LIN {X 0,Y 421.883,Z 601.374,A -85,B 0,C 180,E1 -10153.456,E2 -10153.456} C_VEL
LIN {X 0,Y 421.234,Z 614.501,A -85,B 0,C 180,E1 -10153.897,E2 -10153.897} C_VEL
LIN {X 0,Y 420.74,Z 626.729,A -85,B 0,C 180,E1 -10154.499,E2 -10154.499} C_VEL
LIN {X 0,Y 419.97,Z 639.362,A -85,B 0,C 180,E1 -10155.339,E2 -10155.339} C_VEL
LIN {X 0,Y 419.355,Z 650.7,A -85,B 0,C 180,E1 -10156.307,E2 -10156.307} C_VEL
LIN {X 0,Y 418.794,Z 660.932,A -85,B 0,C 180,E1 -10157.399,E2 -10157.399} C_VEL
LIN {X 0,Y 418.224,Z 670.168,A -85,B 0,C 180,E1 -10158.612,E2 -10158.612} C_VEL
LIN {X 0,Y 417.717,Z 679.182,A -85,B 0,C 180,E1 -10160.07,E2 -10160.07} C_VEL
LIN {X 0,Y 417.45,Z 686.381,A -85,B 0,C 180,E1 -10161.529,E2 -10161.529} C_VEL
LIN {X 0,Y 417.234,Z 692.934,A -85,B 0,C 180,E1 -10163.229,E2 -10163.229} C_VEL
LIN {X 0,Y 417.235,Z 697.222,A -85,B 0,C 180,E1 -10164.685,E2 -10164.685} C_VEL
LIN {X 0,Y 417.147,Z 700.376,A -85,B 0,C 180,E1 -10166.136,E2 -10166.136} C_VEL
LIN {X 0,Y 417.232,Z 701.935,A -85,B 0,C 180,E1 -10167.104,E2 -10167.104} C_VEL
LIN {X 0,Y 417.247,Z 703.007,A -85,B 0,C 180,E1 -10168.07,E2 -10168.07} C_VEL
LIN {X 0,Y 417.206,Z 703.65,A -85,B 0,C 180,E1 -10169.035,E2 -10169.035} C_VEL
LIN {X 0,Y 417.179,Z 703.882,A -85,B 0,C 180,E1 -10170,E2 -10170} C_VEL
LIN {X 0,Y 417.207,Z 703.694,A -85,B 0,C 180,E1 -10170.966,E2 -10170.966} C_VEL
LIN {X 0,Y 417.238,Z 703.046,A -85,B 0,C 180,E1 -10171.931,E2 -10171.931} C_VEL
LIN {X 0,Y 417.242,Z 701.982,A -85,B 0,C 180,E1 -10172.897,E2 -10172.897} C_VEL
LIN {X 0,Y 417.146,Z 700.49,A -85,B 0,C 180,E1 -10173.865,E2 -10173.865} C_VEL
LIN {X 0,Y 417.197,Z 697.385,A -85,B 0,C 180,E1 -10175.317,E2 -10175.317} C_VEL
LIN {X 0,Y 417.243,Z 693.186,A -85,B 0,C 180,E1 -10176.772,E2 -10176.772} C_VEL
LIN {X 0,Y 417.448,Z 686.754,A -85,B 0,C 180,E1 -10178.472,E2 -10178.472} C_VEL
LIN {X 0,Y 417.762,Z 679.755,A -85,B 0,C 180,E1 -10179.93,E2 -10179.93} C_VEL
LIN {X 0,Y 418.247,Z 671.097,A -85,B 0,C 180,E1 -10181.388,E2 -10181.388} C_VEL
LIN {X 0,Y 418.776,Z 662.214,A -85,B 0,C 180,E1 -10182.602,E2 -10182.602} C_VEL
LIN {X 0,Y 419.488,Z 651.309,A -85,B 0,C 180,E1 -10183.813,E2 -10183.813} C_VEL
LIN {X 0,Y 420.239,Z 640.549,A -85,B 0,C 180,E1 -10184.776,E2 -10184.776} C_VEL
LIN {X 0,Y 421.009,Z 628.693,A -85,B 0,C 180,E1 -10185.616,E2 -10185.616} C_VEL
LIN {X 0,Y 421.731,Z 615.268,A -85,B 0,C 180,E1 -10186.333,E2 -10186.333} C_VEL
LIN {X 0,Y 422.424,Z 602.737,A -85,B 0,C 180,E1 -10186.803,E2 -10186.803} C_VEL
LIN {X 0,Y 422.79,Z 586.028,A -85,B 0,C 180,E1 -10187.192,E2 -10187.192} C_VEL
LIN {X 0,Y 423.985,Z 519.859,A -85,B 0,C 180,E1 -10188.527,E2 -10188.527} C_VEL
LIN {X 0,Y 421.419,Z 498.098,A -85,B 0,C 180,E1 -10189.145,E2 -10189.145} C_VEL
LIN {X 0,Y 419.729,Z 487.424,A -85,B 0,C 180,E1 -10189.496,E2 -10189.496} C_VEL
LIN {X 0,Y 420.98,Z 467.923,A -85,B 0,C 180,E1 -10192.98,E2 -10192.98} C_VEL
LIN {X 0,Y 422.264,Z 451.431,A -85,B 0,C 180,E1 -10196.005,E2 -10196.005} C_VEL
LIN {X 0,Y 421.657,Z 446.488,A -85,B 0,C 180,E1 -10197.001,E2 -10197.001} C_VEL
LIN {X 0,Y 419.324,Z 435.566,A -85,B 0,C 180,E1 -10199.362,E2 -10199.362} C_VEL
LIN {X 0,Y 418.269,Z 431.387,A -85,B 0,C 180,E1 -10200.331,E2 -10200.331} C_VEL
LIN {X 0,Y 418.252,Z 431.392,A -85,B 0,C 180,E1 -10203.677,E2 -10203.677} C_VEL
LIN {X 0,Y 418.244,Z 431.39,A -85,B 0,C 180,E1 -10207.224,E2 -10207.224} C_VEL
LIN {X 0,Y 418.255,Z 431.385,A -85,B 0,C 180,E1 -10209.682,E2 -10209.682} C_VEL
LIN {X 0,Y 418.233,Z 431.388,A -85,B 0,C 180,E1 -10212.321,E2 -10212.321} C_VEL
LIN {X 0,Y 418.239,Z 431.387,A -85,B 0,C 180,E1 -10215.109,E2 -10215.109} C_VEL
LIN {X 0,Y 418.238,Z 431.385,A -85,B 0,C 180,E1 -10217.766,E2 -10217.766} C_VEL
LIN {X 0,Y 418.246,Z 431.388,A -85,B 0,C 180,E1 -10220.621,E2 -10220.621} C_VEL
LIN {X 0,Y 418.246,Z 431.384,A -85,B 0,C 180,E1 -10223.976,E2 -10223.976} C_VEL
LIN {X 0,Y 418.261,Z 431.381,A -85,B 0,C 180,E1 -10227.156,E2 -10227.156} C_VEL
LIN {X 0,Y 418.262,Z 431.384,A -85,B 0,C 180,E1 -10230.838,E2 -10230.838} C_VEL
LIN {X 0,Y 418.229,Z 431.388,A -85,B 0,C 180,E1 -10234.093,E2 -10234.093} C_VEL
LIN {X 0,Y 418.231,Z 431.387,A -85,B 0,C 180,E1 -10237.263,E2 -10237.263} C_VEL
LIN {X 0,Y 418.248,Z 431.388,A -85,B 0,C 180,E1 -10240.362,E2 -10240.362} C_VEL
LIN {X 0,Y 418.283,Z 431.381,A -85,B 0,C 180,E1 -10243.403,E2 -10243.403} C_VEL
LIN {X 0,Y 418.348,Z 431.374,A -85,B 0,C 180,E1 -10247.385,E2 -10247.385} C_VEL
LIN {X 0,Y 418.369,Z 431.373,A -85,B 0,C 180,E1 -10251.304,E2 -10251.304} C_VEL
LIN {X 0,Y 418.445,Z 431.365,A -85,B 0,C 180,E1 -10254.518,E2 -10254.518} C_VEL
LIN {X 0,Y 418.966,Z 434.693,A -85,B 0,C 180,E1 -10255.568,E2 -10255.568} C_VEL
LIN {X 0,Y 424.854,Z 448.746,A -85,B 0,C 180,E1 -10256.248,E2 -10256.248} C_VEL
LIN {X 0,Y 423.209,Z 531.742,A -85,B 0,C 180,E1 -10257.952,E2 -10257.952} C_VEL
LIN {X 0,Y 422.943,Z 545.326,A -85,B 0,C 180,E1 -10258.304,E2 -10258.304} C_VEL
LIN {X 0,Y 422.569,Z 558.852,A -85,B 0,C 180,E1 -10258.868,E2 -10258.868} C_VEL
LIN {X 0,Y 422.136,Z 570.169,A -85,B 0,C 180,E1 -10259.519,E2 -10259.519} C_VEL
LIN {X 0,Y 421.493,Z 580.942,A -85,B 0,C 180,E1 -10260.312,E2 -10260.312} C_VEL
LIN {X 0,Y 420.713,Z 592.908,A -85,B 0,C 180,E1 -10261.436,E2 -10261.436} C_VEL
LIN {X 0,Y 420.173,Z 601.191,A -85,B 0,C 180,E1 -10262.397,E2 -10262.397} C_VEL
LIN {X 0,Y 419.534,Z 609.83,A -85,B 0,C 180,E1 -10263.602,E2 -10263.602} C_VEL
LIN {X 0,Y 418.92,Z 618.208,A -85,B 0,C 180,E1 -10265.053,E2 -10265.053} C_VEL
LIN {X 0,Y 418.49,Z 624.908,A -85,B 0,C 180,E1 -10266.509,E2 -10266.509} C_VEL
LIN {X 0,Y 418.087,Z 629.473,A -85,B 0,C 180,E1 -10267.728,E2 -10267.728} C_VEL
LIN {X 0,Y 417.78,Z 633.809,A -85,B 0,C 180,E1 -10269.196,E2 -10269.196} C_VEL
LIN {X 0,Y 417.51,Z 637.049,A -85,B 0,C 180,E1 -10270.671,E2 -10270.671} C_VEL
LIN {X 0,Y 417.341,Z 639.511,A -85,B 0,C 180,E1 -10272.386,E2 -10272.386} C_VEL
LIN {X 0,Y 417.209,Z 640.47,A -85,B 0,C 180,E1 -10273.641,E2 -10273.641} C_VEL
LIN {X 0,Y 417.175,Z 640.732,A -85,B 0,C 180,E1 -10274.637,E2 -10274.637} C_VEL
LIN {X 0,Y 417.198,Z 640.252,A -85,B 0,C 180,E1 -10276.216,E2 -10276.216} C_VEL
LIN {X 0,Y 417.235,Z 638.852,A -85,B 0,C 180,E1 -10277.65,E2 -10277.65} C_VEL
LIN {X 0,Y 417.336,Z 637.328,A -85,B 0,C 180,E1 -10278.661,E2 -10278.661} C_VEL
LIN {X 0,Y 417.508,Z 634.078,A -85,B 0,C 180,E1 -10280.187,E2 -10280.187} C_VEL
LIN {X 0,Y 417.735,Z 629.594,A -85,B 0,C 180,E1 -10281.724,E2 -10281.724} C_VEL
LIN {X 0,Y 418.055,Z 623.72,A -85,B 0,C 180,E1 -10283.27,E2 -10283.27} C_VEL
LIN {X 0,Y 418.516,Z 616.248,A -85,B 0,C 180,E1 -10284.823,E2 -10284.823} C_VEL
LIN {X 0,Y 418.986,Z 608.45,A -85,B 0,C 180,E1 -10286.124,E2 -10286.124} C_VEL
LIN {X 0,Y 419.606,Z 598.921,A -85,B 0,C 180,E1 -10287.414,E2 -10287.414} C_VEL
LIN {X 0,Y 420.198,Z 588.06,A -85,B 0,C 180,E1 -10288.605,E2 -10288.605} C_VEL
LIN {X 0,Y 420.853,Z 576.14,A -85,B 0,C 180,E1 -10289.63,E2 -10289.63} C_VEL
LIN {X 0,Y 421.373,Z 564.13,A -85,B 0,C 180,E1 -10290.439,E2 -10290.439} C_VEL
LIN {X 0,Y 421.814,Z 551.719,A -85,B 0,C 180,E1 -10291.063,E2 -10291.063} C_VEL
LIN {X 0,Y 422.135,Z 538.458,A -85,B 0,C 180,E1 -10291.523,E2 -10291.523} C_VEL
LIN {X 0,Y 422.624,Z 503.985,A -85,B 0,C 180,E1 -10292.209,E2 -10292.209} C_VEL
LIN {X 0,Y 423.54,Z 447.206,A -85,B 0,C 180,E1 -10293.307,E2 -10293.307} C_VEL
LIN {X 0,Y 418.282,Z 431.382,A -85,B 0,C 180,E1 -10293.868,E2 -10293.868} C_VEL
LIN {X 0,Y 418.237,Z 431.383,A -85,B 0,C 180,E1 -10297.225,E2 -10297.225} C_VEL
LIN {X 0,Y 418.21,Z 431.389,A -85,B 0,C 180,E1 -10300.867,E2 -10300.867} C_VEL
LIN {X 0,Y 418.206,Z 431.388,A -85,B 0,C 180,E1 -10303.728,E2 -10303.728} C_VEL
LIN {X 0,Y 418.202,Z 431.395,A -85,B 0,C 180,E1 -10306.447,E2 -10306.447} C_VEL
LIN {X 0,Y 418.209,Z 431.387,A -85,B 0,C 180,E1 -10309.133,E2 -10309.133} C_VEL
LIN {X 0,Y 418.235,Z 431.387,A -85,B 0,C 180,E1 -10312.775,E2 -10312.775} C_VEL
LIN {X 0,Y 418.25,Z 431.388,A -85,B 0,C 180,E1 -10316.323,E2 -10316.323} C_VEL
LIN {X 0,Y 418.243,Z 431.383,A -85,B 0,C 180,E1 -10319.727,E2 -10319.727} C_VEL
LIN {X 0,Y 418.219,Z 431.387,A -85,B 0,C 180,E1 -10323.017,E2 -10323.017} C_VEL
LIN {X 0,Y 418.286,Z 431.382,A -85,B 0,C 180,E1 -10326.218,E2 -10326.218} C_VEL
LIN {X 0,Y 418.252,Z 431.381,A -85,B 0,C 180,E1 -10329.337,E2 -10329.337} C_VEL
LIN {X 0,Y 418.279,Z 431.385,A -85,B 0,C 180,E1 -10332.395,E2 -10332.395} C_VEL
LIN {X 0,Y 418.3,Z 431.375,A -85,B 0,C 180,E1 -10335.403,E2 -10335.403} C_VEL
LIN {X 0,Y 418.316,Z 431.38,A -85,B 0,C 180,E1 -10338.369,E2 -10338.369} C_VEL
LIN {X 0,Y 418.379,Z 431.366,A -85,B 0,C 180,E1 -10341.304,E2 -10341.304} C_VEL
LIN {X 0,Y 418.491,Z 431.356,A -85,B 0,C 180,E1 -10344.217,E2 -10344.217} C_VEL
LIN {X 0,Y 418.366,Z 431.367,A -85,B 0,C 180,E1 -10344.893,E2 -10344.893} C_VEL
LIN {X 0,Y 417.623,Z 431.461,A -85,B 0,C 180,E1 -10345.697,E2 -10345.697} C_VEL
LIN {X 0,Y 414.751,Z 431.821,A -85,B 0,C 180,E1 -10347.005,E2 -10347.005} C_VEL
LIN {X 0,Y 412.417,Z 432.112,A -85,B 0,C 180,E1 -10348.061,E2 -10348.061} C_VEL
LIN {X 0,Y 411.491,Z 432.227,A -85,B 0,C 180,E1 -10348.877,E2 -10348.877} C_VEL
LIN {X 0,Y 411.452,Z 432.229,A -85,B 0,C 180,E1 -10349.152,E2 -10349.152} C_VEL
LIN {X 0,Y 411.635,Z 432.208,A -85,B 0,C 180,E1 -10350,E2 -10350} C_VEL
LIN {X 0,Y 411.446,Z 432.232,A -85,B 0,C 180,E1 -10352.937,E2 -10352.937} C_VEL
LIN {X 0,Y 411.47,Z 432.227,A -85,B 0,C 180,E1 -10355.882,E2 -10355.882} C_VEL
LIN {X 0,Y 411.319,Z 432.248,A -85,B 0,C 180,E1 -10358.846,E2 -10358.846} C_VEL
LIN {X 0,Y 411.284,Z 432.25,A -85,B 0,C 180,E1 -10361.832,E2 -10361.832} C_VEL
LIN {X 0,Y 411.261,Z 432.256,A -85,B 0,C 180,E1 -10364.852,E2 -10364.852} C_VEL
LIN {X 0,Y 411.247,Z 432.255,A -85,B 0,C 180,E1 -10367.915,E2 -10367.915} C_VEL
LIN {X 0,Y 411.197,Z 432.262,A -85,B 0,C 180,E1 -10371.034,E2 -10371.034} C_VEL
LIN {X 0,Y 411.212,Z 432.262,A -85,B 0,C 180,E1 -10374.216,E2 -10374.216} C_VEL
LIN {X 0,Y 411.189,Z 432.261,A -85,B 0,C 180,E1 -10377.482,E2 -10377.482} C_VEL
LIN {X 0,Y 411.189,Z 432.265,A -85,B 0,C 180,E1 -10380.847,E2 -10380.847} C_VEL
LIN {X 0,Y 411.205,Z 432.264,A -85,B 0,C 180,E1 -10384.333,E2 -10384.333} C_VEL
LIN {X 0,Y 411.185,Z 432.263,A -85,B 0,C 180,E1 -10387.974,E2 -10387.974} C_VEL
LIN {X 0,Y 411.157,Z 432.266,A -85,B 0,C 180,E1 -10391.227,E2 -10391.227} C_VEL
LIN {X 0,Y 411.174,Z 432.27,A -85,B 0,C 180,E1 -10394.49,E2 -10394.49} C_VEL
LIN {X 0,Y 411.172,Z 432.266,A -85,B 0,C 180,E1 -10398.194,E2 -10398.194} C_VEL
LIN {X 0,Y 411.209,Z 432.264,A -85,B 0,C 180,E1 -10400.775,E2 -10400.775} C_VEL
LIN {X 0,Y 411.196,Z 432.266,A -85,B 0,C 180,E1 -10404.471,E2 -10404.471} C_VEL
LIN {X 0,Y 411.206,Z 432.263,A -85,B 0,C 180,E1 -10406.873,E2 -10406.873} C_VEL
LIN {X 0,Y 411.232,Z 432.263,A -85,B 0,C 180,E1 -10410.644,E2 -10410.644} C_VEL
LIN {X 0,Y 411.233,Z 432.256,A -85,B 0,C 180,E1 -10413.619,E2 -10413.619} C_VEL
LIN {X 0,Y 411.201,Z 432.264,A -85,B 0,C 180,E1 -10416.852,E2 -10416.852} C_VEL
LIN {X 0,Y 411.214,Z 432.26,A -85,B 0,C 180,E1 -10420.05,E2 -10420.05} C_VEL
LIN {X 0,Y 411.262,Z 432.254,A -85,B 0,C 180,E1 -10423.131,E2 -10423.131} C_VEL
LIN {X 0,Y 411.305,Z 432.251,A -85,B 0,C 180,E1 -10426.896,E2 -10426.896} C_VEL
LIN {X 0,Y 411.291,Z 432.251,A -85,B 0,C 180,E1 -10430.161,E2 -10430.161} C_VEL
LIN {X 0,Y 411.429,Z 432.233,A -85,B 0,C 180,E1 -10433.133,E2 -10433.133} C_VEL
LIN {X 0,Y 411.457,Z 432.23,A -85,B 0,C 180,E1 -10437.063,E2 -10437.063} C_VEL
LIN {X 0,Y 411.64,Z 432.206,A -85,B 0,C 180,E1 -10440,E2 -10440} C_VEL
LIN {X 0,Y 411.463,Z 432.231,A -85,B 0,C 180,E1 -10442.937,E2 -10442.937} C_VEL
LIN {X 0,Y 411.46,Z 432.232,A -85,B 0,C 180,E1 -10446.867,E2 -10446.867} C_VEL
LIN {X 0,Y 411.354,Z 432.246,A -85,B 0,C 180,E1 -10448.845,E2 -10448.845} C_VEL
LIN {X 0,Y 411.283,Z 432.25,A -85,B 0,C 180,E1 -10451.833,E2 -10451.833} C_VEL
LIN {X 0,Y 411.26,Z 432.258,A -85,B 0,C 180,E1 -10454.853,E2 -10454.853} C_VEL
LIN {X 0,Y 411.25,Z 432.254,A -85,B 0,C 180,E1 -10457.915,E2 -10457.915} C_VEL
LIN {X 0,Y 411.196,Z 432.264,A -85,B 0,C 180,E1 -10461.034,E2 -10461.034} C_VEL
LIN {X 0,Y 411.212,Z 432.26,A -85,B 0,C 180,E1 -10464.216,E2 -10464.216} C_VEL
LIN {X 0,Y 411.258,Z 432.253,A -85,B 0,C 180,E1 -10467.478,E2 -10467.478} C_VEL
LIN {X 0,Y 411.189,Z 432.267,A -85,B 0,C 180,E1 -10470.848,E2 -10470.848} C_VEL
LIN {X 0,Y 411.206,Z 432.262,A -85,B 0,C 180,E1 -10474.334,E2 -10474.334} C_VEL
LIN {X 0,Y 411.193,Z 432.261,A -85,B 0,C 180,E1 -10477.974,E2 -10477.974} C_VEL
LIN {X 0,Y 411.163,Z 432.266,A -85,B 0,C 180,E1 -10481.229,E2 -10481.229} C_VEL
LIN {X 0,Y 411.177,Z 432.267,A -85,B 0,C 180,E1 -10484.49,E2 -10484.49} C_VEL
LIN {X 0,Y 411.179,Z 432.264,A -85,B 0,C 180,E1 -10488.195,E2 -10488.195} C_VEL
LIN {X 0,Y 411.22,Z 432.265,A -85,B 0,C 180,E1 -10490.776,E2 -10490.776} C_VEL
LIN {X 0,Y 411.198,Z 432.264,A -85,B 0,C 180,E1 -10494.472,E2 -10494.472} C_VEL
LIN {X 0,Y 411.208,Z 432.265,A -85,B 0,C 180,E1 -10496.874,E2 -10496.874} C_VEL
LIN {X 0,Y 411.252,Z 432.429,A -85,B 0,C 180,E1 -10500.115,E2 -10500.115} C_VEL
LIN {X 0,Y 414.378,Z 446.99,A -85,B 0,C 180,E1 -10503.02,E2 -10503.02} C_VEL
LIN {X 0,Y 415.073,Z 451.482,A -85,B 0,C 180,E1 -10503.882,E2 -10503.882} C_VEL
LIN {X 0,Y 413.777,Z 470.403,A -85,B 0,C 180,E1 -10507.269,E2 -10507.269} C_VEL
LIN {X 0,Y 412.632,Z 489.251,A -85,B 0,C 180,E1 -10510.602,E2 -10510.602} C_VEL
LIN {X 0,Y 412.564,Z 490.802,A -85,B 0,C 180,E1 -10510.858,E2 -10510.858} C_VEL
LIN {X 0,Y 416.226,Z 521.185,A -85,B 0,C 180,E1 -10511.633,E2 -10511.633} C_VEL
LIN {X 0,Y 414.984,Z 601.15,A -85,B 0,C 180,E1 -10513.236,E2 -10513.236} C_VEL
LIN {X 0,Y 414.325,Z 614.166,A -85,B 0,C 180,E1 -10513.684,E2 -10513.684} C_VEL
LIN {X 0,Y 413.798,Z 626.332,A -85,B 0,C 180,E1 -10514.295,E2 -10514.295} C_VEL
LIN {X 0,Y 413.11,Z 638.15,A -85,B 0,C 180,E1 -10515.09,E2 -10515.09} C_VEL
LIN {X 0,Y 412.41,Z 649.606,A -85,B 0,C 180,E1 -10516.072,E2 -10516.072} C_VEL
LIN {X 0,Y 411.839,Z 659.979,A -85,B 0,C 180,E1 -10517.183,E2 -10517.183} C_VEL
LIN {X 0,Y 411.23,Z 669.291,A -85,B 0,C 180,E1 -10518.416,E2 -10518.416} C_VEL
LIN {X 0,Y 410.665,Z 678.366,A -85,B 0,C 180,E1 -10519.897,E2 -10519.897} C_VEL
LIN {X 0,Y 410.372,Z 685.642,A -85,B 0,C 180,E1 -10521.382,E2 -10521.382} C_VEL
LIN {X 0,Y 410.166,Z 692.244,A -85,B 0,C 180,E1 -10523.112,E2 -10523.112} C_VEL
LIN {X 0,Y 410.139,Z 696.57,A -85,B 0,C 180,E1 -10524.592,E2 -10524.592} C_VEL
LIN {X 0,Y 410.061,Z 699.76,A -85,B 0,C 180,E1 -10526.069,E2 -10526.069} C_VEL
LIN {X 0,Y 410.161,Z 701.338,A -85,B 0,C 180,E1 -10527.054,E2 -10527.054} C_VEL
LIN {X 0,Y 410.167,Z 702.433,A -85,B 0,C 180,E1 -10528.037,E2 -10528.037} C_VEL
LIN {X 0,Y 410.152,Z 703.088,A -85,B 0,C 180,E1 -10529.019,E2 -10529.019} C_VEL
LIN {X 0,Y 410.123,Z 703.33,A -85,B 0,C 180,E1 -10530,E2 -10530} C_VEL
LIN {X 0,Y 410.152,Z 703.157,A -85,B 0,C 180,E1 -10530.982,E2 -10530.982} C_VEL
LIN {X 0,Y 410.159,Z 702.518,A -85,B 0,C 180,E1 -10531.964,E2 -10531.964} C_VEL
LIN {X 0,Y 410.17,Z 701.457,A -85,B 0,C 180,E1 -10532.947,E2 -10532.947} C_VEL
LIN {X 0,Y 410.055,Z 699.972,A -85,B 0,C 180,E1 -10533.931,E2 -10533.931} C_VEL
LIN {X 0,Y 410.109,Z 696.884,A -85,B 0,C 180,E1 -10535.409,E2 -10535.409} C_VEL
LIN {X 0,Y 410.175,Z 692.708,A -85,B 0,C 180,E1 -10536.889,E2 -10536.889} C_VEL
LIN {X 0,Y 410.37,Z 686.312,A -85,B 0,C 180,E1 -10538.619,E2 -10538.619} C_VEL
LIN {X 0,Y 410.699,Z 679.327,A -85,B 0,C 180,E1 -10540.102,E2 -10540.102} C_VEL
LIN {X 0,Y 411.24,Z 670.681,A -85,B 0,C 180,E1 -10541.584,E2 -10541.584} C_VEL
LIN {X 0,Y 411.831,Z 661.838,A -85,B 0,C 180,E1 -10542.818,E2 -10542.818} C_VEL
LIN {X 0,Y 412.583,Z 650.958,A -85,B 0,C 180,E1 -10544.049,E2 -10544.049} C_VEL
LIN {X 0,Y 413.366,Z 640.28,A -85,B 0,C 180,E1 -10545.028,E2 -10545.028} C_VEL
LIN {X 0,Y 414.173,Z 628.619,A -85,B 0,C 180,E1 -10545.88,E2 -10545.88} C_VEL
LIN {X 0,Y 414.94,Z 615.447,A -85,B 0,C 180,E1 -10546.608,E2 -10546.608} C_VEL
LIN {X 0,Y 415.703,Z 602.49,A -85,B 0,C 180,E1 -10547.114,E2 -10547.114} C_VEL
LIN {X 0,Y 416.077,Z 587.638,A -85,B 0,C 180,E1 -10547.479,E2 -10547.479} C_VEL
LIN {X 0,Y 417.361,Z 520.325,A -85,B 0,C 180,E1 -10548.87,E2 -10548.87} C_VEL
LIN {X 0,Y 414.842,Z 498.829,A -85,B 0,C 180,E1 -10549.504,E2 -10549.504} C_VEL
LIN {X 0,Y 412.85,Z 486.826,A -85,B 0,C 180,E1 -10549.905,E2 -10549.905} C_VEL
LIN {X 0,Y 414.141,Z 468.177,A -85,B 0,C 180,E1 -10553.309,E2 -10553.309} C_VEL
LIN {X 0,Y 415.43,Z 452.348,A -85,B 0,C 180,E1 -10556.282,E2 -10556.282} C_VEL
LIN {X 0,Y 414.037,Z 444.125,A -85,B 0,C 180,E1 -10558.034,E2 -10558.034} C_VEL
LIN {X 0,Y 411.771,Z 434.506,A -85,B 0,C 180,E1 -10560.232,E2 -10560.232} C_VEL
LIN {X 0,Y 411.228,Z 432.267,A -85,B 0,C 180,E1 -10560.774,E2 -10560.774} C_VEL
LIN {X 0,Y 411.21,Z 432.27,A -85,B 0,C 180,E1 -10564.334,E2 -10564.334} C_VEL
LIN {X 0,Y 411.199,Z 432.264,A -85,B 0,C 180,E1 -10567.974,E2 -10567.974} C_VEL
LIN {X 0,Y 411.185,Z 432.268,A -85,B 0,C 180,E1 -10570.504,E2 -10570.504} C_VEL
LIN {X 0,Y 411.177,Z 432.268,A -85,B 0,C 180,E1 -10573.134,E2 -10573.134} C_VEL
LIN {X 0,Y 411.171,Z 432.265,A -85,B 0,C 180,E1 -10575.881,E2 -10575.881} C_VEL
LIN {X 0,Y 411.164,Z 432.269,A -85,B 0,C 180,E1 -10578.772,E2 -10578.772} C_VEL
LIN {X 0,Y 411.193,Z 432.264,A -85,B 0,C 180,E1 -10582.026,E2 -10582.026} C_VEL
LIN {X 0,Y 411.209,Z 432.258,A -85,B 0,C 180,E1 -10585.667,E2 -10585.667} C_VEL
LIN {X 0,Y 411.192,Z 432.262,A -85,B 0,C 180,E1 -10589.152,E2 -10589.152} C_VEL
LIN {X 0,Y 411.179,Z 432.264,A -85,B 0,C 180,E1 -10591.407,E2 -10591.407} C_VEL
LIN {X 0,Y 411.215,Z 432.262,A -85,B 0,C 180,E1 -10594.934,E2 -10594.934} C_VEL
LIN {X 0,Y 411.201,Z 432.264,A -85,B 0,C 180,E1 -10597.913,E2 -10597.913} C_VEL
LIN {X 0,Y 411.181,Z 432.264,A -85,B 0,C 180,E1 -10601.049,E2 -10601.049} C_VEL
LIN {X 0,Y 411.198,Z 432.266,A -85,B 0,C 180,E1 -10604.129,E2 -10604.129} C_VEL
LIN {X 0,Y 411.298,Z 432.251,A -85,B 0,C 180,E1 -10607.165,E2 -10607.165} C_VEL
LIN {X 0,Y 411.276,Z 432.257,A -85,B 0,C 180,E1 -10610.161,E2 -10610.161} C_VEL
LIN {X 0,Y 411.389,Z 432.243,A -85,B 0,C 180,E1 -10613.132,E2 -10613.132} C_VEL
LIN {X 0,Y 411.445,Z 432.417,A -85,B 0,C 180,E1 -10614.179,E2 -10614.179} C_VEL
LIN {X 0,Y 411.967,Z 435.417,A -85,B 0,C 180,E1 -10615.127,E2 -10615.127} C_VEL
LIN {X 0,Y 418.444,Z 450.705,A -85,B 0,C 180,E1 -10615.906,E2 -10615.906} C_VEL
LIN {X 0,Y 416.337,Z 541.743,A -85,B 0,C 180,E1 -10617.853,E2 -10617.853} C_VEL
LIN {X 0,Y 415.998,Z 555.524,A -85,B 0,C 180,E1 -10618.366,E2 -10618.366} C_VEL
LIN {X 0,Y 415.534,Z 567.804,A -85,B 0,C 180,E1 -10619.031,E2 -10619.031} C_VEL
LIN {X 0,Y 414.856,Z 579.725,A -85,B 0,C 180,E1 -10619.878,E2 -10619.878} C_VEL
LIN {X 0,Y 414.172,Z 590.369,A -85,B 0,C 180,E1 -10620.839,E2 -10620.839} C_VEL
LIN {X 0,Y 413.385,Z 600.255,A -85,B 0,C 180,E1 -10621.948,E2 -10621.948} C_VEL
LIN {X 0,Y 412.753,Z 609.096,A -85,B 0,C 180,E1 -10623.172,E2 -10623.172} C_VEL
LIN {X 0,Y 412.061,Z 617.765,A -85,B 0,C 180,E1 -10624.647,E2 -10624.647} C_VEL
LIN {X 0,Y 411.568,Z 624.674,A -85,B 0,C 180,E1 -10626.127,E2 -10626.127} C_VEL
LIN {X 0,Y 411.034,Z 631.006,A -85,B 0,C 180,E1 -10627.862,E2 -10627.862} C_VEL
LIN {X 0,Y 410.713,Z 635.126,A -85,B 0,C 180,E1 -10629.356,E2 -10629.356} C_VEL
LIN {X 0,Y 410.421,Z 638.158,A -85,B 0,C 180,E1 -10630.857,E2 -10630.857} C_VEL
LIN {X 0,Y 410.274,Z 640.264,A -85,B 0,C 180,E1 -10632.468,E2 -10632.468} C_VEL
LIN {X 0,Y 410.118,Z 641.166,A -85,B 0,C 180,E1 -10633.881,E2 -10633.881} C_VEL
LIN {X 0,Y 410.094,Z 641.305,A -85,B 0,C 180,E1 -10634.896,E2 -10634.896} C_VEL
LIN {X 0,Y 410.134,Z 640.716,A -85,B 0,C 180,E1 -10636.339,E2 -10636.339} C_VEL
LIN {X 0,Y 410.188,Z 638.99,A -85,B 0,C 180,E1 -10637.963,E2 -10637.963} C_VEL
LIN {X 0,Y 410.4,Z 635.97,A -85,B 0,C 180,E1 -10639.632,E2 -10639.632} C_VEL
LIN {X 0,Y 410.56,Z 632.336,A -85,B 0,C 180,E1 -10641.068,E2 -10641.068} C_VEL
LIN {X 0,Y 410.843,Z 626.718,A -85,B 0,C 180,E1 -10642.741,E2 -10642.741} C_VEL
LIN {X 0,Y 411.239,Z 620.397,A -85,B 0,C 180,E1 -10644.215,E2 -10644.215} C_VEL
LIN {X 0,Y 411.739,Z 613.425,A -85,B 0,C 180,E1 -10645.531,E2 -10645.531} C_VEL
LIN {X 0,Y 412.25,Z 604.839,A -85,B 0,C 180,E1 -10646.857,E2 -10646.857} C_VEL
LIN {X 0,Y 412.816,Z 595.717,A -85,B 0,C 180,E1 -10648.009,E2 -10648.009} C_VEL
LIN {X 0,Y 413.452,Z 584.961,A -85,B 0,C 180,E1 -10649.116,E2 -10649.116} C_VEL
LIN {X 0,Y 414,Z 573.904,A -85,B 0,C 180,E1 -10650.029,E2 -10650.029} C_VEL
LIN {X 0,Y 414.543,Z 562.12,A -85,B 0,C 180,E1 -10650.783,E2 -10650.783} C_VEL
LIN {X 0,Y 415.016,Z 548.35,A -85,B 0,C 180,E1 -10651.434,E2 -10651.434} C_VEL
LIN {X 0,Y 415.301,Z 535.233,A -85,B 0,C 180,E1 -10651.84,E2 -10651.84} C_VEL
LIN {X 0,Y 416.605,Z 448.205,A -85,B 0,C 180,E1 -10653.569,E2 -10653.569} C_VEL
LIN {X 0,Y 411.259,Z 432.258,A -85,B 0,C 180,E1 -10654.133,E2 -10654.133} C_VEL
LIN {X 0,Y 411.185,Z 432.264,A -85,B 0,C 180,E1 -10657.975,E2 -10657.975} C_VEL
LIN {X 0,Y 411.151,Z 432.266,A -85,B 0,C 180,E1 -10661.226,E2 -10661.226} C_VEL
LIN {X 0,Y 411.176,Z 432.269,A -85,B 0,C 180,E1 -10664.491,E2 -10664.491} C_VEL
LIN {X 0,Y 411.162,Z 432.269,A -85,B 0,C 180,E1 -10668.192,E2 -10668.192} C_VEL
LIN {X 0,Y 411.192,Z 432.262,A -85,B 0,C 180,E1 -10671.834,E2 -10671.834} C_VEL
LIN {X 0,Y 411.211,Z 432.259,A -85,B 0,C 180,E1 -10675.122,E2 -10675.122} C_VEL
LIN {X 0,Y 411.168,Z 432.266,A -85,B 0,C 180,E1 -10678.002,E2 -10678.002} C_VEL
LIN {X 0,Y 411.18,Z 432.262,A -85,B 0,C 180,E1 -10681.407,E2 -10681.407} C_VEL
LIN {X 0,Y 411.228,Z 432.258,A -85,B 0,C 180,E1 -10684.929,E2 -10684.929} C_VEL
LIN {X 0,Y 411.208,Z 432.261,A -85,B 0,C 180,E1 -10687.913,E2 -10687.913} C_VEL
LIN {X 0,Y 411.219,Z 432.259,A -85,B 0,C 180,E1 -10691.051,E2 -10691.051} C_VEL
LIN {X 0,Y 411.253,Z 432.257,A -85,B 0,C 180,E1 -10694.131,E2 -10694.131} C_VEL
LIN {X 0,Y 411.305,Z 432.247,A -85,B 0,C 180,E1 -10697.165,E2 -10697.165} C_VEL
LIN {X 0,Y 411.292,Z 432.252,A -85,B 0,C 180,E1 -10700.161,E2 -10700.161} C_VEL
LIN {X 0,Y 411.394,Z 432.236,A -85,B 0,C 180,E1 -10703.132,E2 -10703.132} C_VEL
LIN {X 0,Y 411.302,Z 432.248,A -85,B 0,C 180,E1 -10705.099,E2 -10705.099} C_VEL
LIN {X 0,Y 411.511,Z 432.224,A -85,B 0,C 180,E1 -10708.042,E2 -10708.042} C_VEL
LIN {X 0,Y 411.452,Z 432.229,A -85,B 0,C 180,E1 -10709.152,E2 -10709.152} C_VEL
LIN {X 0,Y 410.894,Z 432.301,A -85,B 0,C 180,E1 -10709.97,E2 -10709.97} C_VEL
LIN {X 0,Y 408.089,Z 432.648,A -85,B 0,C 180,E1 -10711.3,E2 -10711.3} C_VEL
LIN {X 0,Y 405.586,Z 432.965,A -85,B 0,C 180,E1 -10712.373,E2 -10712.373} C_VEL
LIN {X 0,Y 404.418,Z 433.106,A -85,B 0,C 180,E1 -10713.203,E2 -10713.203} C_VEL
LIN {X 0,Y 404.276,Z 433.122,A -85,B 0,C 180,E1 -10713.485,E2 -10713.485} C_VEL
LIN {X 0,Y 404.417,Z 433.107,A -85,B 0,C 180,E1 -10715.985,E2 -10715.985} C_VEL
LIN {X 0,Y 404.267,Z 433.125,A -85,B 0,C 180,E1 -10719.001,E2 -10719.001} C_VEL
LIN {X 0,Y 404.257,Z 433.127,A -85,B 0,C 180,E1 -10722.041,E2 -10722.041} C_VEL
LIN {X 0,Y 404.207,Z 433.132,A -85,B 0,C 180,E1 -10725.118,E2 -10725.118} C_VEL
LIN {X 0,Y 404.205,Z 433.135,A -85,B 0,C 180,E1 -10728.238,E2 -10728.238} C_VEL
LIN {X 0,Y 404.139,Z 433.139,A -85,B 0,C 180,E1 -10731.419,E2 -10731.419} C_VEL
LIN {X 0,Y 404.164,Z 433.142,A -85,B 0,C 180,E1 -10734.666,E2 -10734.666} C_VEL
LIN {X 0,Y 404.131,Z 433.142,A -85,B 0,C 180,E1 -10738.004,E2 -10738.004} C_VEL
LIN {X 0,Y 404.144,Z 433.143,A -85,B 0,C 180,E1 -10740.285,E2 -10740.285} C_VEL
LIN {X 0,Y 404.145,Z 433.139,A -85,B 0,C 180,E1 -10743.812,E2 -10743.812} C_VEL
LIN {X 0,Y 404.134,Z 433.144,A -85,B 0,C 180,E1 -10746.874,E2 -10746.874} C_VEL
LIN {X 0,Y 404.119,Z 433.144,A -85,B 0,C 180,E1 -10750.075,E2 -10750.075} C_VEL
LIN {X 0,Y 404.149,Z 433.14,A -85,B 0,C 180,E1 -10753.083,E2 -10753.083} C_VEL
LIN {X 0,Y 404.147,Z 433.139,A -85,B 0,C 180,E1 -10755.926,E2 -10755.926} C_VEL
LIN {X 0,Y 404.114,Z 433.149,A -85,B 0,C 180,E1 -10758.634,E2 -10758.634} C_VEL
LIN {X 0,Y 404.148,Z 433.138,A -85,B 0,C 180,E1 -10761.493,E2 -10761.493} C_VEL
LIN {X 0,Y 404.183,Z 433.137,A -85,B 0,C 180,E1 -10764.984,E2 -10764.984} C_VEL
LIN {X 0,Y 404.142,Z 433.146,A -85,B 0,C 180,E1 -10768.554,E2 -10768.554} C_VEL
LIN {X 0,Y 404.194,Z 433.134,A -85,B 0,C 180,E1 -10772,E2 -10772} C_VEL
LIN {X 0,Y 404.172,Z 433.136,A -85,B 0,C 180,E1 -10775.334,E2 -10775.334} C_VEL
LIN {X 0,Y 404.159,Z 433.144,A -85,B 0,C 180,E1 -10778.582,E2 -10778.582} C_VEL
LIN {X 0,Y 404.204,Z 433.132,A -85,B 0,C 180,E1 -10781.762,E2 -10781.762} C_VEL
LIN {X 0,Y 404.205,Z 433.135,A -85,B 0,C 180,E1 -10784.882,E2 -10784.882} C_VEL
LIN {X 0,Y 404.256,Z 433.126,A -85,B 0,C 180,E1 -10787.959,E2 -10787.959} C_VEL
LIN {X 0,Y 404.402,Z 433.109,A -85,B 0,C 180,E1 -10792.131,E2 -10792.131} C_VEL
LIN {X 0,Y 404.276,Z 433.125,A -85,B 0,C 180,E1 -10795.014,E2 -10795.014} C_VEL
LIN {X 0,Y 404.48,Z 433.098,A -85,B 0,C 180,E1 -10798.009,E2 -10798.009} C_VEL
LIN {X 0,Y 404.609,Z 433.082,A -85,B 0,C 180,E1 -10800,E2 -10800} C_VEL
LIN {X 0,Y 404.42,Z 433.108,A -85,B 0,C 180,E1 -10802.988,E2 -10802.988} C_VEL
LIN {X 0,Y 404.411,Z 433.109,A -85,B 0,C 180,E1 -10806.987,E2 -10806.987} C_VEL
LIN {X 0,Y 404.257,Z 433.126,A -85,B 0,C 180,E1 -10810.012,E2 -10810.012} C_VEL
LIN {X 0,Y 404.266,Z 433.125,A -85,B 0,C 180,E1 -10813.211,E2 -10813.211} C_VEL
LIN {X 0,Y 404.215,Z 433.133,A -85,B 0,C 180,E1 -10817.007,E2 -10817.007} C_VEL
LIN {X 0,Y 404.163,Z 433.14,A -85,B 0,C 180,E1 -10820.352,E2 -10820.352} C_VEL
LIN {X 0,Y 404.16,Z 433.137,A -85,B 0,C 180,E1 -10823.575,E2 -10823.575} C_VEL
LIN {X 0,Y 404.181,Z 433.134,A -85,B 0,C 180,E1 -10825.767,E2 -10825.767} C_VEL
LIN {X 0,Y 404.195,Z 433.133,A -85,B 0,C 180,E1 -10828,E2 -10828} C_VEL
LIN {X 0,Y 404.139,Z 433.14,A -85,B 0,C 180,E1 -10831.558,E2 -10831.558} C_VEL
LIN {X 0,Y 404.184,Z 433.138,A -85,B 0,C 180,E1 -10835.016,E2 -10835.016} C_VEL
LIN {X 0,Y 404.152,Z 433.145,A -85,B 0,C 180,E1 -10838.757,E2 -10838.757} C_VEL
LIN {X 0,Y 404.123,Z 433.142,A -85,B 0,C 180,E1 -10841.6,E2 -10841.6} C_VEL
LIN {X 0,Y 404.146,Z 433.143,A -85,B 0,C 180,E1 -10844.523,E2 -10844.523} C_VEL
LIN {X 0,Y 404.139,Z 433.141,A -85,B 0,C 180,E1 -10847.296,E2 -10847.296} C_VEL
LIN {X 0,Y 404.169,Z 433.136,A -85,B 0,C 180,E1 -10849.956,E2 -10849.956} C_VEL
LIN {X 0,Y 404.136,Z 433.143,A -85,B 0,C 180,E1 -10853.125,E2 -10853.125} C_VEL
LIN {X 0,Y 404.145,Z 433.14,A -85,B 0,C 180,E1 -10856.188,E2 -10856.188} C_VEL
LIN {X 0,Y 404.185,Z 433.2,A -85,B 0,C 180,E1 -10859.847,E2 -10859.847} C_VEL
LIN {X 0,Y 407.3,Z 447.682,A -85,B 0,C 180,E1 -10862.79,E2 -10862.79} C_VEL
LIN {X 0,Y 408.125,Z 452.51,A -85,B 0,C 180,E1 -10863.737,E2 -10863.737} C_VEL
LIN {X 0,Y 406.794,Z 471.109,A -85,B 0,C 180,E1 -10867.125,E2 -10867.125} C_VEL
LIN {X 0,Y 405.681,Z 488.511,A -85,B 0,C 180,E1 -10870.256,E2 -10870.256} C_VEL
LIN {X 0,Y 405.595,Z 490.138,A -85,B 0,C 180,E1 -10870.548,E2 -10870.548} C_VEL
LIN {X 0,Y 409.388,Z 520.876,A -85,B 0,C 180,E1 -10871.366,E2 -10871.366} C_VEL
LIN {X 0,Y 408.078,Z 600.607,A -85,B 0,C 180,E1 -10873.008,E2 -10873.008} C_VEL
LIN {X 0,Y 407.425,Z 613.604,A -85,B 0,C 180,E1 -10873.464,E2 -10873.464} C_VEL
LIN {X 0,Y 406.878,Z 625.779,A -85,B 0,C 180,E1 -10874.085,E2 -10874.085} C_VEL
LIN {X 0,Y 406.238,Z 636.82,A -85,B 0,C 180,E1 -10874.831,E2 -10874.831} C_VEL
LIN {X 0,Y 405.495,Z 648.424,A -85,B 0,C 180,E1 -10875.83,E2 -10875.83} C_VEL
LIN {X 0,Y 404.853,Z 658.936,A -85,B 0,C 180,E1 -10876.958,E2 -10876.958} C_VEL
LIN {X 0,Y 404.232,Z 668.369,A -85,B 0,C 180,E1 -10878.213,E2 -10878.213} C_VEL
LIN {X 0,Y 403.61,Z 677.515,A -85,B 0,C 180,E1 -10879.719,E2 -10879.719} C_VEL
LIN {X 0,Y 403.303,Z 684.878,A -85,B 0,C 180,E1 -10881.23,E2 -10881.23} C_VEL
LIN {X 0,Y 403.136,Z 689.826,A -85,B 0,C 180,E1 -10882.487,E2 -10882.487} C_VEL
LIN {X 0,Y 402.992,Z 694.596,A -85,B 0,C 180,E1 -10883.994,E2 -10883.994} C_VEL
LIN {X 0,Y 402.997,Z 698.197,A -85,B 0,C 180,E1 -10885.499,E2 -10885.499} C_VEL
LIN {X 0,Y 403.092,Z 700.728,A -85,B 0,C 180,E1 -10887.002,E2 -10887.002} C_VEL
LIN {X 0,Y 403.089,Z 701.852,A -85,B 0,C 180,E1 -10888.002,E2 -10888.002} C_VEL
LIN {X 0,Y 403.098,Z 702.522,A -85,B 0,C 180,E1 -10889.001,E2 -10889.001} C_VEL
LIN {X 0,Y 403.069,Z 702.775,A -85,B 0,C 180,E1 -10890,E2 -10890} C_VEL
LIN {X 0,Y 403.099,Z 702.618,A -85,B 0,C 180,E1 -10890.999,E2 -10890.999} C_VEL
LIN {X 0,Y 403.082,Z 701.997,A -85,B 0,C 180,E1 -10891.999,E2 -10891.999} C_VEL
LIN {X 0,Y 403.081,Z 700.948,A -85,B 0,C 180,E1 -10892.999,E2 -10892.999} C_VEL
LIN {X 0,Y 402.969,Z 699.47,A -85,B 0,C 180,E1 -10894.001,E2 -10894.001} C_VEL
LIN {X 0,Y 403.004,Z 696.398,A -85,B 0,C 180,E1 -10895.504,E2 -10895.504} C_VEL
LIN {X 0,Y 403.087,Z 692.238,A -85,B 0,C 180,E1 -10897.011,E2 -10897.011} C_VEL
LIN {X 0,Y 403.282,Z 686.892,A -85,B 0,C 180,E1 -10898.519,E2 -10898.519} C_VEL
LIN {X 0,Y 403.589,Z 680.189,A -85,B 0,C 180,E1 -10900.029,E2 -10900.029} C_VEL
LIN {X 0,Y 404.15,Z 671.833,A -85,B 0,C 180,E1 -10901.536,E2 -10901.536} C_VEL
LIN {X 0,Y 404.689,Z 663.379,A -85,B 0,C 180,E1 -10902.793,E2 -10902.793} C_VEL
LIN {X 0,Y 405.474,Z 653.118,A -85,B 0,C 180,E1 -10904.044,E2 -10904.044} C_VEL
LIN {X 0,Y 406.391,Z 641.605,A -85,B 0,C 180,E1 -10905.163,E2 -10905.163} C_VEL
LIN {X 0,Y 407.233,Z 630.424,A -85,B 0,C 180,E1 -10906.03,E2 -10906.03} C_VEL
LIN {X 0,Y 408.053,Z 618.199,A -85,B 0,C 180,E1 -10906.768,E2 -10906.768} C_VEL
LIN {X 0,Y 408.8,Z 605.687,A -85,B 0,C 180,E1 -10907.316,E2 -10907.316} C_VEL
LIN {X 0,Y 409.288,Z 592.096,A -85,B 0,C 180,E1 -10907.714,E2 -10907.714} C_VEL
LIN {X 0,Y 410.754,Z 520.609,A -85,B 0,C 180,E1 -10909.239,E2 -10909.239} C_VEL
LIN {X 0,Y 408.325,Z 499.878,A -85,B 0,C 180,E1 -10909.876,E2 -10909.876} C_VEL
LIN {X 0,Y 406.017,Z 486.018,A -85,B 0,C 180,E1 -10910.373,E2 -10910.373} C_VEL
LIN {X 0,Y 407.429,Z 467.161,A -85,B 0,C 180,E1 -10913.903,E2 -10913.903} C_VEL
LIN {X 0,Y 408.605,Z 454.323,A -85,B 0,C 180,E1 -10916.368,E2 -10916.368} C_VEL
LIN {X 0,Y 407.694,Z 447.943,A -85,B 0,C 180,E1 -10917.739,E2 -10917.739} C_VEL
LIN {X 0,Y 405.241,Z 437.379,A -85,B 0,C 180,E1 -10920.195,E2 -10920.195} C_VEL
LIN {X 0,Y 404.157,Z 433.148,A -85,B 0,C 180,E1 -10921.3,E2 -10921.3} C_VEL
LIN {X 0,Y 404.149,Z 433.149,A -85,B 0,C 180,E1 -10923.812,E2 -10923.812} C_VEL
LIN {X 0,Y 404.14,Z 433.147,A -85,B 0,C 180,E1 -10926.875,E2 -10926.875} C_VEL
LIN {X 0,Y 404.151,Z 433.143,A -85,B 0,C 180,E1 -10930.08,E2 -10930.08} C_VEL
LIN {X 0,Y 404.156,Z 433.143,A -85,B 0,C 180,E1 -10933.084,E2 -10933.084} C_VEL
LIN {X 0,Y 404.151,Z 433.14,A -85,B 0,C 180,E1 -10935.926,E2 -10935.926} C_VEL
LIN {X 0,Y 404.119,Z 433.148,A -85,B 0,C 180,E1 -10938.635,E2 -10938.635} C_VEL
LIN {X 0,Y 404.152,Z 433.139,A -85,B 0,C 180,E1 -10941.493,E2 -10941.493} C_VEL
LIN {X 0,Y 404.188,Z 433.135,A -85,B 0,C 180,E1 -10944.984,E2 -10944.984} C_VEL
LIN {X 0,Y 404.146,Z 433.145,A -85,B 0,C 180,E1 -10948.554,E2 -10948.554} C_VEL
LIN {X 0,Y 404.155,Z 433.141,A -85,B 0,C 180,E1 -10950.863,E2 -10950.863} C_VEL
LIN {X 0,Y 404.14,Z 433.144,A -85,B 0,C 180,E1 -10954.23,E2 -10954.23} C_VEL
LIN {X 0,Y 404.168,Z 433.139,A -85,B 0,C 180,E1 -10957.508,E2 -10957.508} C_VEL
LIN {X 0,Y 404.134,Z 433.143,A -85,B 0,C 180,E1 -10960.706,E2 -10960.706} C_VEL
LIN {X 0,Y 404.173,Z 433.142,A -85,B 0,C 180,E1 -10963.846,E2 -10963.846} C_VEL
LIN {X 0,Y 404.268,Z 433.127,A -85,B 0,C 180,E1 -10966.938,E2 -10966.938} C_VEL
LIN {X 0,Y 404.244,Z 433.133,A -85,B 0,C 180,E1 -10969.988,E2 -10969.988} C_VEL
LIN {X 0,Y 404.34,Z 433.121,A -85,B 0,C 180,E1 -10973.011,E2 -10973.011} C_VEL
LIN {X 0,Y 404.371,Z 433.229,A -85,B 0,C 180,E1 -10973.701,E2 -10973.701} C_VEL
LIN {X 0,Y 404.992,Z 436.13,A -85,B 0,C 180,E1 -10974.648,E2 -10974.648} C_VEL
LIN {X 0,Y 411.941,Z 452.938,A -85,B 0,C 180,E1 -10975.55,E2 -10975.55} C_VEL
LIN {X 0,Y 409.713,Z 542.197,A -85,B 0,C 180,E1 -10977.511,E2 -10977.511} C_VEL
LIN {X 0,Y 409.338,Z 555.929,A -85,B 0,C 180,E1 -10978.032,E2 -10978.032} C_VEL
LIN {X 0,Y 408.924,Z 567.242,A -85,B 0,C 180,E1 -10978.646,E2 -10978.646} C_VEL
LIN {X 0,Y 408.212,Z 578.769,A -85,B 0,C 180,E1 -10979.453,E2 -10979.453} C_VEL
LIN {X 0,Y 407.435,Z 590.362,A -85,B 0,C 180,E1 -10980.494,E2 -10980.494} C_VEL
LIN {X 0,Y 406.745,Z 599.28,A -85,B 0,C 180,E1 -10981.485,E2 -10981.485} C_VEL
LIN {X 0,Y 406.053,Z 608.424,A -85,B 0,C 180,E1 -10982.728,E2 -10982.728} C_VEL
LIN {X 0,Y 405.25,Z 617.321,A -85,B 0,C 180,E1 -10984.227,E2 -10984.227} C_VEL
LIN {X 0,Y 404.663,Z 624.466,A -85,B 0,C 180,E1 -10985.731,E2 -10985.731} C_VEL
LIN {X 0,Y 404.248,Z 629.275,A -85,B 0,C 180,E1 -10986.99,E2 -10986.99} C_VEL
LIN {X 0,Y 403.85,Z 633.927,A -85,B 0,C 180,E1 -10988.506,E2 -10988.506} C_VEL
LIN {X 0,Y 403.518,Z 637.457,A -85,B 0,C 180,E1 -10990.03,E2 -10990.03} C_VEL
LIN {X 0,Y 403.339,Z 639.214,A -85,B 0,C 180,E1 -10991.05,E2 -10991.05} C_VEL
LIN {X 0,Y 403.191,Z 640.975,A -85,B 0,C 180,E1 -10992.541,E2 -10992.541} C_VEL
LIN {X 0,Y 403.055,Z 641.818,A -85,B 0,C 180,E1 -10994.13,E2 -10994.13} C_VEL
LIN {X 0,Y 403.025,Z 641.787,A -85,B 0,C 180,E1 -10995.163,E2 -10995.163} C_VEL
LIN {X 0,Y 403.068,Z 641.151,A -85,B 0,C 180,E1 -10996.463,E2 -10996.463} C_VEL
LIN {X 0,Y 403.133,Z 639.029,A -85,B 0,C 180,E1 -10998.288,E2 -10998.288} C_VEL
LIN {X 0,Y 403.339,Z 636.205,A -85,B 0,C 180,E1 -10999.791,E2 -10999.791} C_VEL
LIN {X 0,Y 403.537,Z 631.865,A -85,B 0,C 180,E1 -11001.453,E2 -11001.453} C_VEL
LIN {X 0,Y 403.864,Z 626.394,A -85,B 0,C 180,E1 -11003.039,E2 -11003.039} C_VEL
LIN {X 0,Y 404.346,Z 619.233,A -85,B 0,C 180,E1 -11004.655,E2 -11004.655} C_VEL
LIN {X 0,Y 404.816,Z 611.843,A -85,B 0,C 180,E1 -11006,E2 -11006} C_VEL
LIN {X 0,Y 405.456,Z 602.798,A -85,B 0,C 180,E1 -11007.344,E2 -11007.344} C_VEL
LIN {X 0,Y 405.997,Z 592.674,A -85,B 0,C 180,E1 -11008.568,E2 -11008.568} C_VEL
LIN {X 0,Y 406.736,Z 581.495,A -85,B 0,C 180,E1 -11009.644,E2 -11009.644} C_VEL
LIN {X 0,Y 407.316,Z 569.421,A -85,B 0,C 180,E1 -11010.568,E2 -11010.568} C_VEL
LIN {X 0,Y 407.826,Z 557.178,A -85,B 0,C 180,E1 -11011.275,E2 -11011.275} C_VEL
LIN {X 0,Y 408.233,Z 544.128,A -85,B 0,C 180,E1 -11011.818,E2 -11011.818} C_VEL
LIN {X 0,Y 408.446,Z 531.187,A -85,B 0,C 180,E1 -11012.163,E2 -11012.163} C_VEL
LIN {X 0,Y 409.828,Z 449.65,A -85,B 0,C 180,E1 -11013.815,E2 -11013.815} C_VEL
LIN {X 0,Y 404.211,Z 433.136,A -85,B 0,C 180,E1 -11014.412,E2 -11014.412} C_VEL
LIN {X 0,Y 404.137,Z 433.14,A -85,B 0,C 180,E1 -11017.492,E2 -11017.492} C_VEL
LIN {X 0,Y 404.119,Z 433.145,A -85,B 0,C 180,E1 -11020.074,E2 -11020.074} C_VEL
LIN {X 0,Y 404.147,Z 433.139,A -85,B 0,C 180,E1 -11023.082,E2 -11023.082} C_VEL
LIN {X 0,Y 404.146,Z 433.141,A -85,B 0,C 180,E1 -11025.925,E2 -11025.925} C_VEL
LIN {X 0,Y 404.104,Z 433.148,A -85,B 0,C 180,E1 -11028.632,E2 -11028.632} C_VEL
LIN {X 0,Y 404.139,Z 433.139,A -85,B 0,C 180,E1 -11031.495,E2 -11031.495} C_VEL
LIN {X 0,Y 404.185,Z 433.135,A -85,B 0,C 180,E1 -11034.983,E2 -11034.983} C_VEL
LIN {X 0,Y 404.142,Z 433.147,A -85,B 0,C 180,E1 -11038.442,E2 -11038.442} C_VEL
LIN {X 0,Y 404.154,Z 433.14,A -85,B 0,C 180,E1 -11040.862,E2 -11040.862} C_VEL
LIN {X 0,Y 404.146,Z 433.143,A -85,B 0,C 180,E1 -11044.231,E2 -11044.231} C_VEL
LIN {X 0,Y 404.172,Z 433.135,A -85,B 0,C 180,E1 -11047.508,E2 -11047.508} C_VEL
LIN {X 0,Y 404.163,Z 433.141,A -85,B 0,C 180,E1 -11050.707,E2 -11050.707} C_VEL
LIN {X 0,Y 404.221,Z 433.13,A -85,B 0,C 180,E1 -11053.848,E2 -11053.848} C_VEL
LIN {X 0,Y 404.285,Z 433.123,A -85,B 0,C 180,E1 -11056.939,E2 -11056.939} C_VEL
LIN {X 0,Y 404.258,Z 433.127,A -85,B 0,C 180,E1 -11059.988,E2 -11059.988} C_VEL
LIN {X 0,Y 404.344,Z 433.115,A -85,B 0,C 180,E1 -11063.011,E2 -11063.011} C_VEL
LIN {X 0,Y 404.272,Z 433.124,A -85,B 0,C 180,E1 -11065.013,E2 -11065.013} C_VEL
LIN {X 0,Y 404.48,Z 433.099,A -85,B 0,C 180,E1 -11068.008,E2 -11068.008} C_VEL
LIN {X 0,Y 404.604,Z 433.083,A -85,B 0,C 180,E1 -11070,E2 -11070} C_VEL
LIN {X 0,Y 404.404,Z 433.108,A -85,B 0,C 180,E1 -11072.988,E2 -11072.988} C_VEL
LIN {X 0,Y 404.276,Z 433.122,A -85,B 0,C 180,E1 -11073.485,E2 -11073.485} C_VEL
LIN {X 0,Y 403.513,Z 433.223,A -85,B 0,C 180,E1 -11074.316,E2 -11074.316} C_VEL
LIN {X 0,Y 400.732,Z 433.564,A -85,B 0,C 180,E1 -11075.671,E2 -11075.671} C_VEL
LIN {X 0,Y 398.431,Z 433.855,A -85,B 0,C 180,E1 -11076.765,E2 -11076.765} C_VEL
LIN {X 0,Y 397.42,Z 433.977,A -85,B 0,C 180,E1 -11077.609,E2 -11077.609} C_VEL
LIN {X 0,Y 397.32,Z 433.99,A -85,B 0,C 180,E1 -11077.895,E2 -11077.895} C_VEL
LIN {X 0,Y 397.198,Z 434.005,A -85,B 0,C 180,E1 -11081.223,E2 -11081.223} C_VEL
LIN {X 0,Y 397.177,Z 434.012,A -85,B 0,C 180,E1 -11084.343,E2 -11084.343} C_VEL
LIN {X 0,Y 397.145,Z 434.011,A -85,B 0,C 180,E1 -11087.508,E2 -11087.508} C_VEL
LIN {X 0,Y 397.103,Z 434.021,A -85,B 0,C 180,E1 -11090.73,E2 -11090.73} C_VEL
LIN {X 0,Y 397.124,Z 434.015,A -85,B 0,C 180,E1 -11094.018,E2 -11094.018} C_VEL
LIN {X 0,Y 397.102,Z 434.016,A -85,B 0,C 180,E1 -11097.397,E2 -11097.397} C_VEL
LIN {X 0,Y 397.078,Z 434.022,A -85,B 0,C 180,E1 -11100.882,E2 -11100.882} C_VEL
LIN {X 0,Y 397.125,Z 434.02,A -85,B 0,C 180,E1 -11104.493,E2 -11104.493} C_VEL
LIN {X 0,Y 397.092,Z 434.021,A -85,B 0,C 180,E1 -11108.276,E2 -11108.276} C_VEL
LIN {X 0,Y 397.06,Z 434.023,A -85,B 0,C 180,E1 -11111.978,E2 -11111.978} C_VEL
LIN {X 0,Y 397.086,Z 434.02,A -85,B 0,C 180,E1 -11115.069,E2 -11115.069} C_VEL
LIN {X 0,Y 397.061,Z 434.023,A -85,B 0,C 180,E1 -11118.022,E2 -11118.022} C_VEL
LIN {X 0,Y 397.125,Z 434.015,A -85,B 0,C 180,E1 -11121.139,E2 -11121.139} C_VEL
LIN {X 0,Y 397.118,Z 434.02,A -85,B 0,C 180,E1 -11124.497,E2 -11124.497} C_VEL
LIN {X 0,Y 397.078,Z 434.02,A -85,B 0,C 180,E1 -11127.928,E2 -11127.928} C_VEL
LIN {X 0,Y 397.12,Z 434.014,A -85,B 0,C 180,E1 -11131.456,E2 -11131.456} C_VEL
LIN {X 0,Y 397.15,Z 434.016,A -85,B 0,C 180,E1 -11134.488,E2 -11134.488} C_VEL
LIN {X 0,Y 397.108,Z 434.018,A -85,B 0,C 180,E1 -11138.182,E2 -11138.182} C_VEL
LIN {X 0,Y 397.157,Z 434.009,A -85,B 0,C 180,E1 -11141.426,E2 -11141.426} C_VEL
LIN {X 0,Y 397.178,Z 434.014,A -85,B 0,C 180,E1 -11144.608,E2 -11144.608} C_VEL
LIN {X 0,Y 397.219,Z 434.002,A -85,B 0,C 180,E1 -11147.742,E2 -11147.742} C_VEL
LIN {X 0,Y 397.251,Z 434.002,A -85,B 0,C 180,E1 -11150.838,E2 -11150.838} C_VEL
LIN {X 0,Y 397.333,Z 433.992,A -85,B 0,C 180,E1 -11152.888,E2 -11152.888} C_VEL
LIN {X 0,Y 397.247,Z 434.002,A -85,B 0,C 180,E1 -11154.925,E2 -11154.925} C_VEL
LIN {X 0,Y 397.449,Z 433.974,A -85,B 0,C 180,E1 -11157.973,E2 -11157.973} C_VEL
LIN {X 0,Y 397.578,Z 433.958,A -85,B 0,C 180,E1 -11160,E2 -11160} C_VEL
LIN {X 0,Y 397.378,Z 433.985,A -85,B 0,C 180,E1 -11163.041,E2 -11163.041} C_VEL
LIN {X 0,Y 397.364,Z 433.986,A -85,B 0,C 180,E1 -11167.112,E2 -11167.112} C_VEL
LIN {X 0,Y 397.217,Z 434.004,A -85,B 0,C 180,E1 -11170.191,E2 -11170.191} C_VEL
LIN {X 0,Y 397.226,Z 434.002,A -85,B 0,C 180,E1 -11173.321,E2 -11173.321} C_VEL
LIN {X 0,Y 397.181,Z 434.008,A -85,B 0,C 180,E1 -11177.155,E2 -11177.155} C_VEL
LIN {X 0,Y 397.102,Z 434.023,A -85,B 0,C 180,E1 -11180.73,E2 -11180.73} C_VEL
LIN {X 0,Y 397.126,Z 434.014,A -85,B 0,C 180,E1 -11184.019,E2 -11184.019} C_VEL
LIN {X 0,Y 397.193,Z 434.005,A -85,B 0,C 180,E1 -11187.39,E2 -11187.39} C_VEL
LIN {X 0,Y 397.079,Z 434.024,A -85,B 0,C 180,E1 -11190.883,E2 -11190.883} C_VEL
LIN {X 0,Y 397.125,Z 434.018,A -85,B 0,C 180,E1 -11194.494,E2 -11194.494} C_VEL
LIN {X 0,Y 397.101,Z 434.018,A -85,B 0,C 180,E1 -11198.275,E2 -11198.275} C_VEL
LIN {X 0,Y 397.088,Z 434.023,A -85,B 0,C 180,E1 -11200.909,E2 -11200.909} C_VEL
LIN {X 0,Y 397.101,Z 434.016,A -85,B 0,C 180,E1 -11203.649,E2 -11203.649} C_VEL
LIN {X 0,Y 397.105,Z 434.02,A -85,B 0,C 180,E1 -11206.521,E2 -11206.521} C_VEL
LIN {X 0,Y 397.114,Z 434.018,A -85,B 0,C 180,E1 -11210.423,E2 -11210.423} C_VEL
LIN {X 0,Y 397.108,Z 434.017,A -85,B 0,C 180,E1 -11214.266,E2 -11214.266} C_VEL
LIN {X 0,Y 397.115,Z 434.021,A -85,B 0,C 180,E1 -11216.728,E2 -11216.728} C_VEL
LIN {X 0,Y 397.133,Z 434.115,A -85,B 0,C 180,E1 -11219.605,E2 -11219.605} C_VEL
LIN {X 0,Y 400.215,Z 448.337,A -85,B 0,C 180,E1 -11222.551,E2 -11222.551} C_VEL
LIN {X 0,Y 401.18,Z 454.126,A -85,B 0,C 180,E1 -11223.704,E2 -11223.704} C_VEL
LIN {X 0,Y 399.6,Z 474.692,A -85,B 0,C 180,E1 -11227.51,E2 -11227.51} C_VEL
LIN {X 0,Y 398.618,Z 489.949,A -85,B 0,C 180,E1 -11230.278,E2 -11230.278} C_VEL
LIN {X 0,Y 402.501,Z 522.21,A -85,B 0,C 180,E1 -11231.14,E2 -11231.14} C_VEL
LIN {X 0,Y 401.185,Z 599.813,A -85,B 0,C 180,E1 -11232.773,E2 -11232.773} C_VEL
LIN {X 0,Y 400.485,Z 613.602,A -85,B 0,C 180,E1 -11233.268,E2 -11233.268} C_VEL
LIN {X 0,Y 399.88,Z 626.104,A -85,B 0,C 180,E1 -11233.93,E2 -11233.93} C_VEL
LIN {X 0,Y 399.078,Z 638.543,A -85,B 0,C 180,E1 -11234.814,E2 -11234.814} C_VEL
LIN {X 0,Y 398.306,Z 650.065,A -85,B 0,C 180,E1 -11235.863,E2 -11235.863} C_VEL
LIN {X 0,Y 397.756,Z 659.864,A -85,B 0,C 180,E1 -11236.981,E2 -11236.981} C_VEL
LIN {X 0,Y 397.1,Z 669.034,A -85,B 0,C 180,E1 -11238.257,E2 -11238.257} C_VEL
LIN {X 0,Y 396.489,Z 677.984,A -85,B 0,C 180,E1 -11239.79,E2 -11239.79} C_VEL
LIN {X 0,Y 396.202,Z 685.111,A -85,B 0,C 180,E1 -11241.328,E2 -11241.328} C_VEL
LIN {X 0,Y 396.005,Z 690.786,A -85,B 0,C 180,E1 -11242.864,E2 -11242.864} C_VEL
LIN {X 0,Y 395.96,Z 695.207,A -85,B 0,C 180,E1 -11244.398,E2 -11244.398} C_VEL
LIN {X 0,Y 395.897,Z 698.481,A -85,B 0,C 180,E1 -11245.928,E2 -11245.928} C_VEL
LIN {X 0,Y 396.023,Z 700.099,A -85,B 0,C 180,E1 -11246.949,E2 -11246.949} C_VEL
LIN {X 0,Y 396.015,Z 701.258,A -85,B 0,C 180,E1 -11247.966,E2 -11247.966} C_VEL
LIN {X 0,Y 396.046,Z 701.949,A -85,B 0,C 180,E1 -11248.984,E2 -11248.984} C_VEL
LIN {X 0,Y 396.016,Z 702.217,A -85,B 0,C 180,E1 -11250,E2 -11250} C_VEL
LIN {X 0,Y 396.029,Z 702.072,A -85,B 0,C 180,E1 -11251.017,E2 -11251.017} C_VEL
LIN {X 0,Y 396.008,Z 701.479,A -85,B 0,C 180,E1 -11252.034,E2 -11252.034} C_VEL
LIN {X 0,Y 395.995,Z 700.439,A -85,B 0,C 180,E1 -11253.052,E2 -11253.052} C_VEL
LIN {X 0,Y 395.886,Z 698.968,A -85,B 0,C 180,E1 -11254.072,E2 -11254.072} C_VEL
LIN {X 0,Y 395.902,Z 695.913,A -85,B 0,C 180,E1 -11255.603,E2 -11255.603} C_VEL
LIN {X 0,Y 396.014,Z 691.769,A -85,B 0,C 180,E1 -11257.137,E2 -11257.137} C_VEL
LIN {X 0,Y 396.201,Z 686.456,A -85,B 0,C 180,E1 -11258.672,E2 -11258.672} C_VEL
LIN {X 0,Y 396.535,Z 679.809,A -85,B 0,C 180,E1 -11260.209,E2 -11260.209} C_VEL
LIN {X 0,Y 397.142,Z 671.521,A -85,B 0,C 180,E1 -11261.743,E2 -11261.743} C_VEL
LIN {X 0,Y 397.75,Z 663.107,A -85,B 0,C 180,E1 -11263.02,E2 -11263.02} C_VEL
LIN {X 0,Y 398.553,Z 652.889,A -85,B 0,C 180,E1 -11264.293,E2 -11264.293} C_VEL
LIN {X 0,Y 399.516,Z 641.483,A -85,B 0,C 180,E1 -11265.431,E2 -11265.431} C_VEL
LIN {X 0,Y 400.416,Z 630.407,A -85,B 0,C 180,E1 -11266.31,E2 -11266.31} C_VEL
LIN {X 0,Y 401.335,Z 617.288,A -85,B 0,C 180,E1 -11267.123,E2 -11267.123} C_VEL
LIN {X 0,Y 402.216,Z 603.916,A -85,B 0,C 180,E1 -11267.707,E2 -11267.707} C_VEL
LIN {X 0,Y 402.709,Z 589.953,A -85,B 0,C 180,E1 -11268.112,E2 -11268.112} C_VEL
LIN {X 0,Y 404.201,Z 521.078,A -85,B 0,C 180,E1 -11269.621,E2 -11269.621} C_VEL
LIN {X 0,Y 401.689,Z 499.903,A -85,B 0,C 180,E1 -11270.297,E2 -11270.297} C_VEL
LIN {X 0,Y 399.24,Z 485.237,A -85,B 0,C 180,E1 -11270.86,E2 -11270.86} C_VEL
LIN {X 0,Y 400.583,Z 467.96,A -85,B 0,C 180,E1 -11274.173,E2 -11274.173} C_VEL
LIN {X 0,Y 401.791,Z 455.45,A -85,B 0,C 180,E1 -11276.635,E2 -11276.635} C_VEL
LIN {X 0,Y 400.238,Z 446.754,A -85,B 0,C 180,E1 -11278.6,E2 -11278.6} C_VEL
LIN {X 0,Y 398.094,Z 437.746,A -85,B 0,C 180,E1 -11280.796,E2 -11280.796} C_VEL
LIN {X 0,Y 397.1,Z 434.028,A -85,B 0,C 180,E1 -11281.786,E2 -11281.786} C_VEL
LIN {X 0,Y 397.129,Z 434.024,A -85,B 0,C 180,E1 -11284.493,E2 -11284.493} C_VEL
LIN {X 0,Y 397.107,Z 434.02,A -85,B 0,C 180,E1 -11288.275,E2 -11288.275} C_VEL
LIN {X 0,Y 397.092,Z 434.023,A -85,B 0,C 180,E1 -11290.909,E2 -11290.909} C_VEL
LIN {X 0,Y 397.104,Z 434.018,A -85,B 0,C 180,E1 -11293.649,E2 -11293.649} C_VEL
LIN {X 0,Y 397.104,Z 434.022,A -85,B 0,C 180,E1 -11296.521,E2 -11296.521} C_VEL
LIN {X 0,Y 397.116,Z 434.021,A -85,B 0,C 180,E1 -11300.423,E2 -11300.423} C_VEL
LIN {X 0,Y 397.111,Z 434.019,A -85,B 0,C 180,E1 -11304.265,E2 -11304.265} C_VEL
LIN {X 0,Y 397.118,Z 434.018,A -85,B 0,C 180,E1 -11306.727,E2 -11306.727} C_VEL
LIN {X 0,Y 397.121,Z 434.017,A -85,B 0,C 180,E1 -11310.295,E2 -11310.295} C_VEL
LIN {X 0,Y 397.086,Z 434.021,A -85,B 0,C 180,E1 -11313.738,E2 -11313.738} C_VEL
LIN {X 0,Y 397.102,Z 434.019,A -85,B 0,C 180,E1 -11317.085,E2 -11317.085} C_VEL
LIN {X 0,Y 397.097,Z 434.023,A -85,B 0,C 180,E1 -11320.35,E2 -11320.35} C_VEL
LIN {X 0,Y 397.118,Z 434.019,A -85,B 0,C 180,E1 -11323.551,E2 -11323.551} C_VEL
LIN {X 0,Y 397.194,Z 434.009,A -85,B 0,C 180,E1 -11326.701,E2 -11326.701} C_VEL
LIN {X 0,Y 397.205,Z 434.01,A -85,B 0,C 180,E1 -11329.809,E2 -11329.809} C_VEL
LIN {X 0,Y 397.322,Z 434.116,A -85,B 0,C 180,E1 -11333.206,E2 -11333.206} C_VEL
LIN {X 0,Y 398.054,Z 437.21,A -85,B 0,C 180,E1 -11334.186,E2 -11334.186} C_VEL
LIN {X 0,Y 405.388,Z 454.26,A -85,B 0,C 180,E1 -11335.148,E2 -11335.148} C_VEL
LIN {X 0,Y 403.319,Z 534.603,A -85,B 0,C 180,E1 -11336.943,E2 -11336.943} C_VEL
LIN {X 0,Y 403.005,Z 547.655,A -85,B 0,C 180,E1 -11337.314,E2 -11337.314} C_VEL
LIN {X 0,Y 402.603,Z 560.291,A -85,B 0,C 180,E1 -11337.874,E2 -11337.874} C_VEL
LIN {X 0,Y 402.024,Z 572.616,A -85,B 0,C 180,E1 -11338.623,E2 -11338.623} C_VEL
LIN {X 0,Y 401.235,Z 583.814,A -85,B 0,C 180,E1 -11339.508,E2 -11339.508} C_VEL
LIN {X 0,Y 400.384,Z 594.665,A -85,B 0,C 180,E1 -11340.591,E2 -11340.591} C_VEL
LIN {X 0,Y 399.638,Z 604.155,A -85,B 0,C 180,E1 -11341.764,E2 -11341.764} C_VEL
LIN {X 0,Y 398.854,Z 612.575,A -85,B 0,C 180,E1 -11343.03,E2 -11343.03} C_VEL
LIN {X 0,Y 398.109,Z 620.749,A -85,B 0,C 180,E1 -11344.556,E2 -11344.556} C_VEL
LIN {X 0,Y 397.531,Z 627.318,A -85,B 0,C 180,E1 -11346.089,E2 -11346.089} C_VEL
LIN {X 0,Y 397.052,Z 632.426,A -85,B 0,C 180,E1 -11347.592,E2 -11347.592} C_VEL
LIN {X 0,Y 396.652,Z 636.568,A -85,B 0,C 180,E1 -11349.176,E2 -11349.176} C_VEL
LIN {X 0,Y 396.443,Z 638.624,A -85,B 0,C 180,E1 -11350.211,E2 -11350.211} C_VEL
LIN {X 0,Y 396.266,Z 640.232,A -85,B 0,C 180,E1 -11351.25,E2 -11351.25} C_VEL
LIN {X 0,Y 396.124,Z 641.676,A -85,B 0,C 180,E1 -11352.627,E2 -11352.627} C_VEL
LIN {X 0,Y 395.966,Z 642.405,A -85,B 0,C 180,E1 -11354.388,E2 -11354.388} C_VEL
LIN {X 0,Y 395.976,Z 642.26,A -85,B 0,C 180,E1 -11355.44,E2 -11355.44} C_VEL
LIN {X 0,Y 396.003,Z 641.563,A -85,B 0,C 180,E1 -11356.592,E2 -11356.592} C_VEL
LIN {X 0,Y 396.026,Z 640.57,A -85,B 0,C 180,E1 -11357.559,E2 -11357.559} C_VEL
LIN {X 0,Y 396.168,Z 638.083,A -85,B 0,C 180,E1 -11359.159,E2 -11359.159} C_VEL
LIN {X 0,Y 396.357,Z 634.454,A -85,B 0,C 180,E1 -11360.771,E2 -11360.771} C_VEL
LIN {X 0,Y 396.651,Z 629.611,A -85,B 0,C 180,E1 -11362.376,E2 -11362.376} C_VEL
LIN {X 0,Y 397.069,Z 623.179,A -85,B 0,C 180,E1 -11364.022,E2 -11364.022} C_VEL
LIN {X 0,Y 397.66,Z 615.018,A -85,B 0,C 180,E1 -11365.664,E2 -11365.664} C_VEL
LIN {X 0,Y 398.187,Z 606.6,A -85,B 0,C 180,E1 -11367.032,E2 -11367.032} C_VEL
LIN {X 0,Y 398.822,Z 597.6,A -85,B 0,C 180,E1 -11368.224,E2 -11368.224} C_VEL
LIN {X 0,Y 399.485,Z 587.024,A -85,B 0,C 180,E1 -11369.367,E2 -11369.367} C_VEL
LIN {X 0,Y 400.096,Z 575.923,A -85,B 0,C 180,E1 -11370.332,E2 -11370.332} C_VEL
LIN {X 0,Y 400.704,Z 563.335,A -85,B 0,C 180,E1 -11371.18,E2 -11371.18} C_VEL
LIN {X 0,Y 401.183,Z 549.719,A -85,B 0,C 180,E1 -11371.853,E2 -11371.853} C_VEL
LIN {X 0,Y 401.488,Z 537.122,A -85,B 0,C 180,E1 -11372.269,E2 -11372.269} C_VEL
LIN {X 0,Y 402.911,Z 450.803,A -85,B 0,C 180,E1 -11374.071,E2 -11374.071} C_VEL
LIN {X 0,Y 397.158,Z 434.014,A -85,B 0,C 180,E1 -11374.695,E2 -11374.695} C_VEL
LIN {X 0,Y 397.092,Z 434.023,A -85,B 0,C 180,E1 -11378.276,E2 -11378.276} C_VEL
LIN {X 0,Y 397.056,Z 434.024,A -85,B 0,C 180,E1 -11381.976,E2 -11381.976} C_VEL
LIN {X 0,Y 397.087,Z 434.019,A -85,B 0,C 180,E1 -11385.069,E2 -11385.069} C_VEL
LIN {X 0,Y 397.054,Z 434.025,A -85,B 0,C 180,E1 -11388.023,E2 -11388.023} C_VEL
LIN {X 0,Y 397.091,Z 434.018,A -85,B 0,C 180,E1 -11391.723,E2 -11391.723} C_VEL
LIN {X 0,Y 397.127,Z 434.013,A -85,B 0,C 180,E1 -11395.506,E2 -11395.506} C_VEL
LIN {X 0,Y 397.08,Z 434.02,A -85,B 0,C 180,E1 -11399.117,E2 -11399.117} C_VEL
LIN {X 0,Y 397.084,Z 434.023,A -85,B 0,C 180,E1 -11402.246,E2 -11402.246} C_VEL
LIN {X 0,Y 397.126,Z 434.015,A -85,B 0,C 180,E1 -11405.981,E2 -11405.981} C_VEL
LIN {X 0,Y 397.141,Z 434.012,A -85,B 0,C 180,E1 -11409.704,E2 -11409.704} C_VEL
LIN {X 0,Y 397.184,Z 434.009,A -85,B 0,C 180,E1 -11412.845,E2 -11412.845} C_VEL
LIN {X 0,Y 397.231,Z 434.004,A -85,B 0,C 180,E1 -11416.702,E2 -11416.702} C_VEL
LIN {X 0,Y 397.218,Z 434.003,A -85,B 0,C 180,E1 -11419.809,E2 -11419.809} C_VEL
LIN {X 0,Y 397.297,Z 433.994,A -85,B 0,C 180,E1 -11422.887,E2 -11422.887} C_VEL
LIN {X 0,Y 397.243,Z 434.001,A -85,B 0,C 180,E1 -11424.925,E2 -11424.925} C_VEL
LIN {X 0,Y 397.448,Z 433.975,A -85,B 0,C 180,E1 -11427.973,E2 -11427.973} C_VEL
LIN {X 0,Y 397.574,Z 433.959,A -85,B 0,C 180,E1 -11430,E2 -11430} C_VEL
LIN {X 0,Y 397.338,Z 433.988,A -85,B 0,C 180,E1 -11433.041,E2 -11433.041} C_VEL
LIN {X 0,Y 397.367,Z 433.986,A -85,B 0,C 180,E1 -11436.091,E2 -11436.091} C_VEL
LIN {X 0,Y 397.32,Z 433.99,A -85,B 0,C 180,E1 -11437.895,E2 -11437.895} C_VEL
LIN {X 0,Y 396.586,Z 434.086,A -85,B 0,C 180,E1 -11438.74,E2 -11438.74} C_VEL
LIN {X 0,Y 393.654,Z 434.448,A -85,B 0,C 180,E1 -11440.112,E2 -11440.112} C_VEL
LIN {X 0,Y 391.228,Z 434.748,A -85,B 0,C 180,E1 -11441.221,E2 -11441.221} C_VEL
LIN {X 0,Y 390.225,Z 434.875,A -85,B 0,C 180,E1 -11442.08,E2 -11442.08} C_VEL
LIN {X 0,Y 390.163,Z 434.886,A -85,B 0,C 180,E1 -11442.37,E2 -11442.37} C_VEL
LIN {X 0,Y 390.14,Z 434.884,A -85,B 0,C 180,E1 -11445.676,E2 -11445.676} C_VEL
LIN {X 0,Y 390.103,Z 434.891,A -85,B 0,C 180,E1 -11448.922,E2 -11448.922} C_VEL
LIN {X 0,Y 390.038,Z 434.9,A -85,B 0,C 180,E1 -11452.234,E2 -11452.234} C_VEL
LIN {X 0,Y 390.084,Z 434.891,A -85,B 0,C 180,E1 -11455.732,E2 -11455.732} C_VEL
LIN {X 0,Y 390.034,Z 434.898,A -85,B 0,C 180,E1 -11459.111,E2 -11459.111} C_VEL
LIN {X 0,Y 390.043,Z 434.901,A -85,B 0,C 180,E1 -11462.721,E2 -11462.721} C_VEL
LIN {X 0,Y 390.055,Z 434.894,A -85,B 0,C 180,E1 -11465.825,E2 -11465.825} C_VEL
LIN {X 0,Y 390.037,Z 434.897,A -85,B 0,C 180,E1 -11469.212,E2 -11469.212} C_VEL
LIN {X 0,Y 390.037,Z 434.901,A -85,B 0,C 180,E1 -11472.373,E2 -11472.373} C_VEL
LIN {X 0,Y 390.043,Z 434.896,A -85,B 0,C 180,E1 -11475.354,E2 -11475.354} C_VEL
LIN {X 0,Y 390.024,Z 434.901,A -85,B 0,C 180,E1 -11478.186,E2 -11478.186} C_VEL
LIN {X 0,Y 390.086,Z 434.893,A -85,B 0,C 180,E1 -11480.907,E2 -11480.907} C_VEL
LIN {X 0,Y 390.084,Z 434.895,A -85,B 0,C 180,E1 -11484.793,E2 -11484.793} C_VEL
LIN {X 0,Y 390.023,Z 434.904,A -85,B 0,C 180,E1 -11488.496,E2 -11488.496} C_VEL
LIN {X 0,Y 390.116,Z 434.888,A -85,B 0,C 180,E1 -11492.07,E2 -11492.07} C_VEL
LIN {X 0,Y 390.076,Z 434.891,A -85,B 0,C 180,E1 -11495.519,E2 -11495.519} C_VEL
LIN {X 0,Y 390.062,Z 434.897,A -85,B 0,C 180,E1 -11498.878,E2 -11498.878} C_VEL
LIN {X 0,Y 390.125,Z 434.887,A -85,B 0,C 180,E1 -11502.167,E2 -11502.167} C_VEL
LIN {X 0,Y 390.143,Z 434.883,A -85,B 0,C 180,E1 -11505.393,E2 -11505.393} C_VEL
LIN {X 0,Y 390.147,Z 434.889,A -85,B 0,C 180,E1 -11508.571,E2 -11508.571} C_VEL
LIN {X 0,Y 390.305,Z 434.864,A -85,B 0,C 180,E1 -11512.034,E2 -11512.034} C_VEL
LIN {X 0,Y 390.217,Z 434.879,A -85,B 0,C 180,E1 -11514.833,E2 -11514.833} C_VEL
LIN {X 0,Y 390.418,Z 434.849,A -85,B 0,C 180,E1 -11517.937,E2 -11517.937} C_VEL
LIN {X 0,Y 390.548,Z 434.833,A -85,B 0,C 180,E1 -11520,E2 -11520} C_VEL
LIN {X 0,Y 390.312,Z 434.864,A -85,B 0,C 180,E1 -11523.097,E2 -11523.097} C_VEL
LIN {X 0,Y 390.33,Z 434.862,A -85,B 0,C 180,E1 -11526.202,E2 -11526.202} C_VEL
LIN {X 0,Y 390.314,Z 434.864,A -85,B 0,C 180,E1 -11528.282,E2 -11528.282} C_VEL
LIN {X 0,Y 390.17,Z 434.884,A -85,B 0,C 180,E1 -11532.483,E2 -11532.483} C_VEL
LIN {X 0,Y 390.139,Z 434.883,A -85,B 0,C 180,E1 -11535.677,E2 -11535.677} C_VEL
LIN {X 0,Y 390.104,Z 434.892,A -85,B 0,C 180,E1 -11538.922,E2 -11538.922} C_VEL
LIN {X 0,Y 390.037,Z 434.898,A -85,B 0,C 180,E1 -11542.234,E2 -11542.234} C_VEL
LIN {X 0,Y 390.117,Z 434.886,A -85,B 0,C 180,E1 -11545.743,E2 -11545.743} C_VEL
LIN {X 0,Y 390.058,Z 434.896,A -85,B 0,C 180,E1 -11549.11,E2 -11549.11} C_VEL
LIN {X 0,Y 390.042,Z 434.903,A -85,B 0,C 180,E1 -11552.722,E2 -11552.722} C_VEL
LIN {X 0,Y 390.056,Z 434.894,A -85,B 0,C 180,E1 -11555.826,E2 -11555.826} C_VEL
LIN {X 0,Y 390.068,Z 434.894,A -85,B 0,C 180,E1 -11559.218,E2 -11559.218} C_VEL
LIN {X 0,Y 390.042,Z 434.899,A -85,B 0,C 180,E1 -11562.374,E2 -11562.374} C_VEL
LIN {X 0,Y 390.047,Z 434.896,A -85,B 0,C 180,E1 -11565.355,E2 -11565.355} C_VEL
LIN {X 0,Y 390.033,Z 434.898,A -85,B 0,C 180,E1 -11568.187,E2 -11568.187} C_VEL
LIN {X 0,Y 390.091,Z 434.895,A -85,B 0,C 180,E1 -11570.908,E2 -11570.908} C_VEL
LIN {X 0,Y 390.085,Z 434.897,A -85,B 0,C 180,E1 -11574.793,E2 -11574.793} C_VEL
LIN {X 0,Y 390.029,Z 434.901,A -85,B 0,C 180,E1 -11578.497,E2 -11578.497} C_VEL
LIN {X 0,Y 390.115,Z 435.07,A -85,B 0,C 180,E1 -11579.37,E2 -11579.37} C_VEL
LIN {X 0,Y 393.381,Z 450.182,A -85,B 0,C 180,E1 -11582.554,E2 -11582.554} C_VEL
LIN {X 0,Y 394.198,Z 454.999,A -85,B 0,C 180,E1 -11583.531,E2 -11583.531} C_VEL
LIN {X 0,Y 392.715,Z 473.892,A -85,B 0,C 180,E1 -11587.093,E2 -11587.093} C_VEL
LIN {X 0,Y 391.668,Z 489.28,A -85,B 0,C 180,E1 -11589.964,E2 -11589.964} C_VEL
LIN {X 0,Y 395.653,Z 522.538,A -85,B 0,C 180,E1 -11590.886,E2 -11590.886} C_VEL
LIN {X 0,Y 394.288,Z 599.014,A -85,B 0,C 180,E1 -11592.529,E2 -11592.529} C_VEL
LIN {X 0,Y 393.6,Z 612.87,A -85,B 0,C 180,E1 -11593.033,E2 -11593.033} C_VEL
LIN {X 0,Y 392.895,Z 625.418,A -85,B 0,C 180,E1 -11593.704,E2 -11593.704} C_VEL
LIN {X 0,Y 392.223,Z 637.113,A -85,B 0,C 180,E1 -11594.542,E2 -11594.542} C_VEL
LIN {X 0,Y 391.532,Z 647.177,A -85,B 0,C 180,E1 -11595.446,E2 -11595.446} C_VEL
LIN {X 0,Y 390.827,Z 657.727,A -85,B 0,C 180,E1 -11596.614,E2 -11596.614} C_VEL
LIN {X 0,Y 390.165,Z 666.351,A -85,B 0,C 180,E1 -11597.781,E2 -11597.781} C_VEL
LIN {X 0,Y 389.566,Z 675.691,A -85,B 0,C 180,E1 -11599.344,E2 -11599.344} C_VEL
LIN {X 0,Y 389.168,Z 683.201,A -85,B 0,C 180,E1 -11600.909,E2 -11600.909} C_VEL
LIN {X 0,Y 389.015,Z 688.27,A -85,B 0,C 180,E1 -11602.213,E2 -11602.213} C_VEL
LIN {X 0,Y 388.874,Z 693.154,A -85,B 0,C 180,E1 -11603.775,E2 -11603.775} C_VEL
LIN {X 0,Y 388.862,Z 696.852,A -85,B 0,C 180,E1 -11605.335,E2 -11605.335} C_VEL
LIN {X 0,Y 388.957,Z 699.469,A -85,B 0,C 180,E1 -11606.893,E2 -11606.893} C_VEL
LIN {X 0,Y 388.943,Z 700.659,A -85,B 0,C 180,E1 -11607.929,E2 -11607.929} C_VEL
LIN {X 0,Y 388.994,Z 701.375,A -85,B 0,C 180,E1 -11608.965,E2 -11608.965} C_VEL
LIN {X 0,Y 388.964,Z 701.658,A -85,B 0,C 180,E1 -11610,E2 -11610} C_VEL
LIN {X 0,Y 388.947,Z 701.525,A -85,B 0,C 180,E1 -11611.036,E2 -11611.036} C_VEL
LIN {X 0,Y 388.936,Z 700.96,A -85,B 0,C 180,E1 -11612.071,E2 -11612.071} C_VEL
LIN {X 0,Y 388.895,Z 699.928,A -85,B 0,C 180,E1 -11613.108,E2 -11613.108} C_VEL
LIN {X 0,Y 388.806,Z 698.474,A -85,B 0,C 180,E1 -11614.147,E2 -11614.147} C_VEL
LIN {X 0,Y 388.805,Z 695.094,A -85,B 0,C 180,E1 -11615.864,E2 -11615.864} C_VEL
LIN {X 0,Y 388.94,Z 691.349,A -85,B 0,C 180,E1 -11617.267,E2 -11617.267} C_VEL
LIN {X 0,Y 389.135,Z 686.061,A -85,B 0,C 180,E1 -11618.831,E2 -11618.831} C_VEL
LIN {X 0,Y 389.485,Z 679.443,A -85,B 0,C 180,E1 -11620.396,E2 -11620.396} C_VEL
LIN {X 0,Y 390.134,Z 671.209,A -85,B 0,C 180,E1 -11621.957,E2 -11621.957} C_VEL
LIN {X 0,Y 390.817,Z 662.829,A -85,B 0,C 180,E1 -11623.255,E2 -11623.255} C_VEL
LIN {X 0,Y 391.647,Z 652.704,A -85,B 0,C 180,E1 -11624.55,E2 -11624.55} C_VEL
LIN {X 0,Y 392.668,Z 641.489,A -85,B 0,C 180,E1 -11625.707,E2 -11625.707} C_VEL
LIN {X 0,Y 393.607,Z 630.62,A -85,B 0,C 180,E1 -11626.6,E2 -11626.6} C_VEL
LIN {X 0,Y 394.581,Z 617.751,A -85,B 0,C 180,E1 -11627.425,E2 -11627.425} C_VEL
LIN {X 0,Y 395.49,Z 604.979,A -85,B 0,C 180,E1 -11628.018,E2 -11628.018} C_VEL
LIN {X 0,Y 396.057,Z 590.692,A -85,B 0,C 180,E1 -11628.46,E2 -11628.46} C_VEL
LIN {X 0,Y 397.712,Z 522.122,A -85,B 0,C 180,E1 -11630.006,E2 -11630.006} C_VEL
LIN {X 0,Y 395.489,Z 502.453,A -85,B 0,C 180,E1 -11630.655,E2 -11630.655} C_VEL
LIN {X 0,Y 392.443,Z 484.653,A -85,B 0,C 180,E1 -11631.339,E2 -11631.339} C_VEL
LIN {X 0,Y 393.788,Z 468.746,A -85,B 0,C 180,E1 -11634.466,E2 -11634.466} C_VEL
LIN {X 0,Y 394.941,Z 457.819,A -85,B 0,C 180,E1 -11636.662,E2 -11636.662} C_VEL
LIN {X 0,Y 394.234,Z 452.309,A -85,B 0,C 180,E1 -11637.902,E2 -11637.902} C_VEL
LIN {X 0,Y 392.216,Z 443.229,A -85,B 0,C 180,E1 -11640.115,E2 -11640.115} C_VEL
LIN {X 0,Y 390.039,Z 434.909,A -85,B 0,C 180,E1 -11642.334,E2 -11642.334} C_VEL
LIN {X 0,Y 390.089,Z 434.9,A -85,B 0,C 180,E1 -11645.207,E2 -11645.207} C_VEL
LIN {X 0,Y 390.074,Z 434.896,A -85,B 0,C 180,E1 -11649.219,E2 -11649.219} C_VEL
LIN {X 0,Y 390.046,Z 434.899,A -85,B 0,C 180,E1 -11652.374,E2 -11652.374} C_VEL
LIN {X 0,Y 390.047,Z 434.897,A -85,B 0,C 180,E1 -11655.355,E2 -11655.355} C_VEL
LIN {X 0,Y 390.031,Z 434.901,A -85,B 0,C 180,E1 -11658.186,E2 -11658.186} C_VEL
LIN {X 0,Y 390.09,Z 434.893,A -85,B 0,C 180,E1 -11660.907,E2 -11660.907} C_VEL
LIN {X 0,Y 390.088,Z 434.893,A -85,B 0,C 180,E1 -11664.793,E2 -11664.793} C_VEL
LIN {X 0,Y 390.027,Z 434.903,A -85,B 0,C 180,E1 -11668.496,E2 -11668.496} C_VEL
LIN {X 0,Y 390.029,Z 434.9,A -85,B 0,C 180,E1 -11672.063,E2 -11672.063} C_VEL
LIN {X 0,Y 390.046,Z 434.899,A -85,B 0,C 180,E1 -11675.517,E2 -11675.517} C_VEL
LIN {X 0,Y 390.051,Z 434.898,A -85,B 0,C 180,E1 -11678.877,E2 -11678.877} C_VEL
LIN {X 0,Y 390.073,Z 434.895,A -85,B 0,C 180,E1 -11682.73,E2 -11682.73} C_VEL
LIN {X 0,Y 390.135,Z 434.889,A -85,B 0,C 180,E1 -11686.601,E2 -11686.601} C_VEL
LIN {X 0,Y 390.157,Z 434.887,A -85,B 0,C 180,E1 -11689.622,E2 -11689.622} C_VEL
LIN {X 0,Y 390.27,Z 434.982,A -85,B 0,C 180,E1 -11692.669,E2 -11692.669} C_VEL
LIN {X 0,Y 390.969,Z 437.919,A -85,B 0,C 180,E1 -11693.646,E2 -11693.646} C_VEL
LIN {X 0,Y 397.374,Z 452.308,A -85,B 0,C 180,E1 -11694.527,E2 -11694.527} C_VEL
LIN {X 0,Y 399.069,Z 456.419,A -85,B 0,C 180,E1 -11694.757,E2 -11694.757} C_VEL
LIN {X 0,Y 396.554,Z 542.797,A -85,B 0,C 180,E1 -11696.762,E2 -11696.762} C_VEL
LIN {X 0,Y 396.162,Z 556.605,A -85,B 0,C 180,E1 -11697.299,E2 -11697.299} C_VEL
LIN {X 0,Y 395.65,Z 568.578,A -85,B 0,C 180,E1 -11697.964,E2 -11697.964} C_VEL
LIN {X 0,Y 394.804,Z 580.699,A -85,B 0,C 180,E1 -11698.852,E2 -11698.852} C_VEL
LIN {X 0,Y 393.988,Z 591.459,A -85,B 0,C 180,E1 -11699.859,E2 -11699.859} C_VEL
LIN {X 0,Y 393.1,Z 601.492,A -85,B 0,C 180,E1 -11701.024,E2 -11701.024} C_VEL
LIN {X 0,Y 392.316,Z 610.416,A -85,B 0,C 180,E1 -11702.31,E2 -11702.31} C_VEL
LIN {X 0,Y 391.422,Z 619.165,A -85,B 0,C 180,E1 -11703.861,E2 -11703.861} C_VEL
LIN {X 0,Y 390.753,Z 626.153,A -85,B 0,C 180,E1 -11705.418,E2 -11705.418} C_VEL
LIN {X 0,Y 390.108,Z 632.531,A -85,B 0,C 180,E1 -11707.245,E2 -11707.245} C_VEL
LIN {X 0,Y 389.705,Z 636.695,A -85,B 0,C 180,E1 -11708.818,E2 -11708.818} C_VEL
LIN {X 0,Y 389.356,Z 639.765,A -85,B 0,C 180,E1 -11710.399,E2 -11710.399} C_VEL
LIN {X 0,Y 389.183,Z 641.253,A -85,B 0,C 180,E1 -11711.457,E2 -11711.457} C_VEL
LIN {X 0,Y 389.049,Z 642.384,A -85,B 0,C 180,E1 -11712.71,E2 -11712.71} C_VEL
LIN {X 0,Y 388.909,Z 642.991,A -85,B 0,C 180,E1 -11714.655,E2 -11714.655} C_VEL
LIN {X 0,Y 388.903,Z 642.662,A -85,B 0,C 180,E1 -11715.728,E2 -11715.728} C_VEL
LIN {X 0,Y 388.929,Z 641.898,A -85,B 0,C 180,E1 -11716.805,E2 -11716.805} C_VEL
LIN {X 0,Y 388.975,Z 640.698,A -85,B 0,C 180,E1 -11717.888,E2 -11717.888} C_VEL
LIN {X 0,Y 389.169,Z 637.964,A -85,B 0,C 180,E1 -11719.517,E2 -11719.517} C_VEL
LIN {X 0,Y 389.365,Z 634.048,A -85,B 0,C 180,E1 -11721.161,E2 -11721.161} C_VEL
LIN {X 0,Y 389.637,Z 629.251,A -85,B 0,C 180,E1 -11722.694,E2 -11722.694} C_VEL
LIN {X 0,Y 390.144,Z 622.079,A -85,B 0,C 180,E1 -11724.476,E2 -11724.476} C_VEL
LIN {X 0,Y 390.696,Z 614.807,A -85,B 0,C 180,E1 -11725.917,E2 -11725.917} C_VEL
LIN {X 0,Y 391.249,Z 606.496,A -85,B 0,C 180,E1 -11727.262,E2 -11727.262} C_VEL
LIN {X 0,Y 391.937,Z 595.956,A -85,B 0,C 180,E1 -11728.643,E2 -11728.643} C_VEL
LIN {X 0,Y 392.663,Z 585.156,A -85,B 0,C 180,E1 -11729.78,E2 -11729.78} C_VEL
LIN {X 0,Y 393.289,Z 573.888,A -85,B 0,C 180,E1 -11730.723,E2 -11730.723} C_VEL
LIN {X 0,Y 393.916,Z 561.418,A -85,B 0,C 180,E1 -11731.532,E2 -11731.532} C_VEL
LIN {X 0,Y 394.333,Z 548.884,A -85,B 0,C 180,E1 -11732.133,E2 -11732.133} C_VEL
LIN {X 0,Y 394.617,Z 535.31,A -85,B 0,C 180,E1 -11732.56,E2 -11732.56} C_VEL
LIN {X 0,Y 396.195,Z 452.612,A -85,B 0,C 180,E1 -11734.313,E2 -11734.313} C_VEL
LIN {X 0,Y 390.135,Z 434.887,A -85,B 0,C 180,E1 -11734.988,E2 -11734.988} C_VEL
LIN {X 0,Y 390.059,Z 434.894,A -85,B 0,C 180,E1 -11739.096,E2 -11739.096} C_VEL
LIN {X 0,Y 390.034,Z 434.904,A -85,B 0,C 180,E1 -11742.372,E2 -11742.372} C_VEL
LIN {X 0,Y 390.044,Z 434.895,A -85,B 0,C 180,E1 -11745.354,E2 -11745.354} C_VEL
LIN {X 0,Y 390.017,Z 434.903,A -85,B 0,C 180,E1 -11748.184,E2 -11748.184} C_VEL
LIN {X 0,Y 390.058,Z 434.895,A -85,B 0,C 180,E1 -11750.903,E2 -11750.903} C_VEL
LIN {X 0,Y 390.086,Z 434.893,A -85,B 0,C 180,E1 -11754.793,E2 -11754.793} C_VEL
LIN {X 0,Y 390.026,Z 434.904,A -85,B 0,C 180,E1 -11758.495,E2 -11758.495} C_VEL
LIN {X 0,Y 390.03,Z 434.9,A -85,B 0,C 180,E1 -11762.063,E2 -11762.063} C_VEL
LIN {X 0,Y 390.056,Z 434.894,A -85,B 0,C 180,E1 -11765.517,E2 -11765.517} C_VEL
LIN {X 0,Y 390.065,Z 434.895,A -85,B 0,C 180,E1 -11768.878,E2 -11768.878} C_VEL
LIN {X 0,Y 390.127,Z 434.889,A -85,B 0,C 180,E1 -11772.166,E2 -11772.166} C_VEL
LIN {X 0,Y 390.144,Z 434.883,A -85,B 0,C 180,E1 -11775.392,E2 -11775.392} C_VEL
LIN {X 0,Y 390.149,Z 434.888,A -85,B 0,C 180,E1 -11778.571,E2 -11778.571} C_VEL
LIN {X 0,Y 390.258,Z 434.871,A -85,B 0,C 180,E1 -11782.085,E2 -11782.085} C_VEL
LIN {X 0,Y 390.213,Z 434.877,A -85,B 0,C 180,E1 -11784.833,E2 -11784.833} C_VEL
LIN {X 0,Y 390.417,Z 434.85,A -85,B 0,C 180,E1 -11787.936,E2 -11787.936} C_VEL
LIN {X 0,Y 390.543,Z 434.835,A -85,B 0,C 180,E1 -11790,E2 -11790} C_VEL
LIN {X 0,Y 390.274,Z 434.868,A -85,B 0,C 180,E1 -11793.096,E2 -11793.096} C_VEL
LIN {X 0,Y 390.32,Z 434.865,A -85,B 0,C 180,E1 -11796.202,E2 -11796.202} C_VEL
LIN {X 0,Y 390.194,Z 434.877,A -85,B 0,C 180,E1 -11799.329,E2 -11799.329} C_VEL
LIN {X 0,Y 390.163,Z 434.886,A -85,B 0,C 180,E1 -11802.37,E2 -11802.37} C_VEL
LIN {X 0,Y 389.53,Z 434.971,A -85,B 0,C 180,E1 -11803.232,E2 -11803.232} C_VEL
LIN {X 0,Y 386.638,Z 435.327,A -85,B 0,C 180,E1 -11804.631,E2 -11804.631} C_VEL
LIN {X 0,Y 384.181,Z 435.626,A -85,B 0,C 180,E1 -11805.761,E2 -11805.761} C_VEL
LIN {X 0,Y 383.153,Z 435.759,A -85,B 0,C 180,E1 -11806.637,E2 -11806.637} C_VEL
LIN {X 0,Y 383.085,Z 435.763,A -85,B 0,C 180,E1 -11806.933,E2 -11806.933} C_VEL
LIN {X 0,Y 383.029,Z 435.775,A -85,B 0,C 180,E1 -11810.647,E2 -11810.647} C_VEL
LIN {X 0,Y 383.017,Z 435.771,A -85,B 0,C 180,E1 -11813.808,E2 -11813.808} C_VEL
LIN {X 0,Y 382.994,Z 435.774,A -85,B 0,C 180,E1 -11817.306,E2 -11817.306} C_VEL
LIN {X 0,Y 382.982,Z 435.778,A -85,B 0,C 180,E1 -11820.918,E2 -11820.918} C_VEL
LIN {X 0,Y 383.017,Z 435.776,A -85,B 0,C 180,E1 -11824.668,E2 -11824.668} C_VEL
LIN {X 0,Y 382.993,Z 435.775,A -85,B 0,C 180,E1 -11827.902,E2 -11827.902} C_VEL
LIN {X 0,Y 382.964,Z 435.778,A -85,B 0,C 180,E1 -11831.35,E2 -11831.35} C_VEL
LIN {X 0,Y 382.994,Z 435.777,A -85,B 0,C 180,E1 -11834.303,E2 -11834.303} C_VEL
LIN {X 0,Y 383.009,Z 435.772,A -85,B 0,C 180,E1 -11837.24,E2 -11837.24} C_VEL
LIN {X 0,Y 383.007,Z 435.777,A -85,B 0,C 180,E1 -11840.415,E2 -11840.415} C_VEL
LIN {X 0,Y 383.023,Z 435.771,A -85,B 0,C 180,E1 -11844.044,E2 -11844.044} C_VEL
LIN {X 0,Y 382.986,Z 435.775,A -85,B 0,C 180,E1 -11847.578,E2 -11847.578} C_VEL
LIN {X 0,Y 382.991,Z 435.777,A -85,B 0,C 180,E1 -11850.3,E2 -11850.3} C_VEL
LIN {X 0,Y 383.078,Z 435.764,A -85,B 0,C 180,E1 -11854.021,E2 -11854.021} C_VEL
LIN {X 0,Y 383.011,Z 435.772,A -85,B 0,C 180,E1 -11857.335,E2 -11857.335} C_VEL
LIN {X 0,Y 383.058,Z 435.772,A -85,B 0,C 180,E1 -11860.716,E2 -11860.716} C_VEL
LIN {X 0,Y 383.08,Z 435.764,A -85,B 0,C 180,E1 -11864.027,E2 -11864.027} C_VEL
LIN {X 0,Y 383.136,Z 435.757,A -85,B 0,C 180,E1 -11867.284,E2 -11867.284} C_VEL
LIN {X 0,Y 383.15,Z 435.76,A -85,B 0,C 180,E1 -11870.498,E2 -11870.498} C_VEL
LIN {X 0,Y 383.241,Z 435.75,A -85,B 0,C 180,E1 -11872.625,E2 -11872.625} C_VEL
LIN {X 0,Y 383.189,Z 435.755,A -85,B 0,C 180,E1 -11874.738,E2 -11874.738} C_VEL
LIN {X 0,Y 383.385,Z 435.725,A -85,B 0,C 180,E1 -11877.899,E2 -11877.899} C_VEL
LIN {X 0,Y 383.517,Z 435.709,A -85,B 0,C 180,E1 -11880,E2 -11880} C_VEL
LIN {X 0,Y 383.248,Z 435.744,A -85,B 0,C 180,E1 -11883.154,E2 -11883.154} C_VEL
LIN {X 0,Y 383.287,Z 435.74,A -85,B 0,C 180,E1 -11886.316,E2 -11886.316} C_VEL
LIN {X 0,Y 383.26,Z 435.745,A -85,B 0,C 180,E1 -11888.436,E2 -11888.436} C_VEL
LIN {X 0,Y 383.096,Z 435.761,A -85,B 0,C 180,E1 -11891.642,E2 -11891.642} C_VEL
LIN {X 0,Y 383.11,Z 435.764,A -85,B 0,C 180,E1 -11894.882,E2 -11894.882} C_VEL
LIN {X 0,Y 383.088,Z 435.764,A -85,B 0,C 180,E1 -11898.172,E2 -11898.172} C_VEL
LIN {X 0,Y 382.992,Z 435.774,A -85,B 0,C 180,E1 -11901.531,E2 -11901.531} C_VEL
LIN {X 0,Y 383.049,Z 435.771,A -85,B 0,C 180,E1 -11904.961,E2 -11904.961} C_VEL
LIN {X 0,Y 383.04,Z 435.772,A -85,B 0,C 180,E1 -11908.493,E2 -11908.493} C_VEL
LIN {X 0,Y 383.009,Z 435.773,A -85,B 0,C 180,E1 -11912.15,E2 -11912.15} C_VEL
LIN {X 0,Y 383.018,Z 435.777,A -85,B 0,C 180,E1 -11914.668,E2 -11914.668} C_VEL
LIN {X 0,Y 382.998,Z 435.773,A -85,B 0,C 180,E1 -11917.904,E2 -11917.904} C_VEL
LIN {X 0,Y 382.983,Z 435.776,A -85,B 0,C 180,E1 -11921.348,E2 -11921.348} C_VEL
LIN {X 0,Y 382.997,Z 435.776,A -85,B 0,C 180,E1 -11924.304,E2 -11924.304} C_VEL
LIN {X 0,Y 383.01,Z 435.773,A -85,B 0,C 180,E1 -11927.241,E2 -11927.241} C_VEL
LIN {X 0,Y 383.016,Z 435.774,A -85,B 0,C 180,E1 -11930.414,E2 -11930.414} C_VEL
LIN {X 0,Y 383.025,Z 435.77,A -85,B 0,C 180,E1 -11934.045,E2 -11934.045} C_VEL
LIN {X 0,Y 382.987,Z 435.775,A -85,B 0,C 180,E1 -11937.578,E2 -11937.578} C_VEL
LIN {X 0,Y 383.013,Z 435.81,A -85,B 0,C 180,E1 -11939.084,E2 -11939.084} C_VEL
LIN {X 0,Y 386.305,Z 451.076,A -85,B 0,C 180,E1 -11942.361,E2 -11942.361} C_VEL
LIN {X 0,Y 387.196,Z 457.089,A -85,B 0,C 180,E1 -11943.596,E2 -11943.596} C_VEL
LIN {X 0,Y 385.606,Z 475.957,A -85,B 0,C 180,E1 -11947.214,E2 -11947.214} C_VEL
LIN {X 0,Y 384.734,Z 488.809,A -85,B 0,C 180,E1 -11949.657,E2 -11949.657} C_VEL
LIN {X 0,Y 388.822,Z 523.461,A -85,B 0,C 180,E1 -11950.632,E2 -11950.632} C_VEL
LIN {X 0,Y 387.37,Z 599.143,A -85,B 0,C 180,E1 -11952.309,E2 -11952.309} C_VEL
LIN {X 0,Y 386.673,Z 612.76,A -85,B 0,C 180,E1 -11952.822,E2 -11952.822} C_VEL
LIN {X 0,Y 385.986,Z 624.673,A -85,B 0,C 180,E1 -11953.471,E2 -11953.471} C_VEL
LIN {X 0,Y 385.218,Z 637.199,A -85,B 0,C 180,E1 -11954.389,E2 -11954.389} C_VEL
LIN {X 0,Y 384.418,Z 648.215,A -85,B 0,C 180,E1 -11955.416,E2 -11955.416} C_VEL
LIN {X 0,Y 383.705,Z 658.637,A -85,B 0,C 180,E1 -11956.63,E2 -11956.63} C_VEL
LIN {X 0,Y 382.97,Z 668.685,A -85,B 0,C 180,E1 -11958.086,E2 -11958.086} C_VEL
LIN {X 0,Y 382.423,Z 676.147,A -85,B 0,C 180,E1 -11959.411,E2 -11959.411} C_VEL
LIN {X 0,Y 382.058,Z 683.473,A -85,B 0,C 180,E1 -11961.005,E2 -11961.005} C_VEL
LIN {X 0,Y 381.861,Z 689.274,A -85,B 0,C 180,E1 -11962.598,E2 -11962.598} C_VEL
LIN {X 0,Y 381.761,Z 693.629,A -85,B 0,C 180,E1 -11964.119,E2 -11964.119} C_VEL
LIN {X 0,Y 381.744,Z 697.169,A -85,B 0,C 180,E1 -11965.777,E2 -11965.777} C_VEL
LIN {X 0,Y 381.872,Z 698.828,A -85,B 0,C 180,E1 -11966.835,E2 -11966.835} C_VEL
LIN {X 0,Y 381.874,Z 700.044,A -85,B 0,C 180,E1 -11967.891,E2 -11967.891} C_VEL
LIN {X 0,Y 381.925,Z 700.794,A -85,B 0,C 180,E1 -11968.946,E2 -11968.946} C_VEL
LIN {X 0,Y 381.914,Z 701.096,A -85,B 0,C 180,E1 -11970,E2 -11970} C_VEL
LIN {X 0,Y 381.868,Z 700.979,A -85,B 0,C 180,E1 -11971.055,E2 -11971.055} C_VEL
LIN {X 0,Y 381.864,Z 700.443,A -85,B 0,C 180,E1 -11972.11,E2 -11972.11} C_VEL
LIN {X 0,Y 381.796,Z 699.434,A -85,B 0,C 180,E1 -11973.166,E2 -11973.166} C_VEL
LIN {X 0,Y 381.727,Z 697.997,A -85,B 0,C 180,E1 -11974.224,E2 -11974.224} C_VEL
LIN {X 0,Y 381.763,Z 696.133,A -85,B 0,C 180,E1 -11975.282,E2 -11975.282} C_VEL
LIN {X 0,Y 381.787,Z 692.422,A -85,B 0,C 180,E1 -11976.872,E2 -11976.872} C_VEL
LIN {X 0,Y 381.995,Z 687.578,A -85,B 0,C 180,E1 -11978.464,E2 -11978.464} C_VEL
LIN {X 0,Y 382.347,Z 681.455,A -85,B 0,C 180,E1 -11980.057,E2 -11980.057} C_VEL
LIN {X 0,Y 382.945,Z 673.841,A -85,B 0,C 180,E1 -11981.647,E2 -11981.647} C_VEL
LIN {X 0,Y 383.68,Z 664.453,A -85,B 0,C 180,E1 -11983.237,E2 -11983.237} C_VEL
LIN {X 0,Y 384.546,Z 654.97,A -85,B 0,C 180,E1 -11984.537,E2 -11984.537} C_VEL
LIN {X 0,Y 385.608,Z 644.199,A -85,B 0,C 180,E1 -11985.731,E2 -11985.731} C_VEL
LIN {X 0,Y 386.66,Z 632.516,A -85,B 0,C 180,E1 -11986.771,E2 -11986.771} C_VEL
LIN {X 0,Y 387.718,Z 620.41,A -85,B 0,C 180,E1 -11987.607,E2 -11987.607} C_VEL
LIN {X 0,Y 388.568,Z 608.811,A -85,B 0,C 180,E1 -11988.214,E2 -11988.214} C_VEL
LIN {X 0,Y 389.328,Z 595.169,A -85,B 0,C 180,E1 -11988.723,E2 -11988.723} C_VEL
LIN {X 0,Y 391.204,Z 522.321,A -85,B 0,C 180,E1 -11990.439,E2 -11990.439} C_VEL
LIN {X 0,Y 388.884,Z 501.913,A -85,B 0,C 180,E1 -11991.138,E2 -11991.138} C_VEL
LIN {X 0,Y 385.67,Z 483.858,A -85,B 0,C 180,E1 -11991.89,E2 -11991.89} C_VEL
LIN {X 0,Y 387.094,Z 468.709,A -85,B 0,C 180,E1 -11994.94,E2 -11994.94} C_VEL
LIN {X 0,Y 388.151,Z 459.15,A -85,B 0,C 180,E1 -11996.915,E2 -11996.915} C_VEL
LIN {X 0,Y 386.922,Z 451.637,A -85,B 0,C 180,E1 -11998.692,E2 -11998.692} C_VEL
LIN {X 0,Y 384.927,Z 443.037,A -85,B 0,C 180,E1 -12000.893,E2 -12000.893} C_VEL
LIN {X 0,Y 382.993,Z 435.786,A -85,B 0,C 180,E1 -12002.932,E2 -12002.932} C_VEL
LIN {X 0,Y 383.036,Z 435.777,A -85,B 0,C 180,E1 -12006.165,E2 -12006.165} C_VEL
LIN {X 0,Y 383.012,Z 435.776,A -85,B 0,C 180,E1 -12009.959,E2 -12009.959} C_VEL
LIN {X 0,Y 383.009,Z 435.778,A -85,B 0,C 180,E1 -12012.779,E2 -12012.779} C_VEL
LIN {X 0,Y 383,Z 435.774,A -85,B 0,C 180,E1 -12015.789,E2 -12015.789} C_VEL
LIN {X 0,Y 382.99,Z 435.778,A -85,B 0,C 180,E1 -12018.796,E2 -12018.796} C_VEL
LIN {X 0,Y 383.001,Z 435.776,A -85,B 0,C 180,E1 -12022.097,E2 -12022.097} C_VEL
LIN {X 0,Y 383.022,Z 435.77,A -85,B 0,C 180,E1 -12025.332,E2 -12025.332} C_VEL
LIN {X 0,Y 382.986,Z 435.776,A -85,B 0,C 180,E1 -12029.082,E2 -12029.082} C_VEL
LIN {X 0,Y 382.985,Z 435.78,A -85,B 0,C 180,E1 -12032.692,E2 -12032.692} C_VEL
LIN {X 0,Y 383.013,Z 435.775,A -85,B 0,C 180,E1 -12036.191,E2 -12036.191} C_VEL
LIN {X 0,Y 383.038,Z 435.771,A -85,B 0,C 180,E1 -12039.597,E2 -12039.597} C_VEL
LIN {X 0,Y 383.041,Z 435.771,A -85,B 0,C 180,E1 -12042.928,E2 -12042.928} C_VEL
LIN {X 0,Y 383.093,Z 435.767,A -85,B 0,C 180,E1 -12046.487,E2 -12046.487} C_VEL
LIN {X 0,Y 383.122,Z 435.763,A -85,B 0,C 180,E1 -12049.43,E2 -12049.43} C_VEL
LIN {X 0,Y 383.261,Z 435.779,A -85,B 0,C 180,E1 -12052.065,E2 -12052.065} C_VEL
LIN {X 0,Y 383.945,Z 438.751,A -85,B 0,C 180,E1 -12053.084,E2 -12053.084} C_VEL
LIN {X 0,Y 390.076,Z 452.029,A -85,B 0,C 180,E1 -12053.96,E2 -12053.96} C_VEL
LIN {X 0,Y 392.692,Z 458.726,A -85,B 0,C 180,E1 -12054.35,E2 -12054.35} C_VEL
LIN {X 0,Y 390.025,Z 544.132,A -85,B 0,C 180,E1 -12056.384,E2 -12056.384} C_VEL
LIN {X 0,Y 389.573,Z 558.303,A -85,B 0,C 180,E1 -12056.962,E2 -12056.962} C_VEL
LIN {X 0,Y 388.982,Z 570.345,A -85,B 0,C 180,E1 -12057.67,E2 -12057.67} C_VEL
LIN {X 0,Y 388.102,Z 582.172,A -85,B 0,C 180,E1 -12058.573,E2 -12058.573} C_VEL
LIN {X 0,Y 387.143,Z 593.724,A -85,B 0,C 180,E1 -12059.704,E2 -12059.704} C_VEL
LIN {X 0,Y 386.062,Z 604.573,A -85,B 0,C 180,E1 -12061.043,E2 -12061.043} C_VEL
LIN {X 0,Y 385.268,Z 613.104,A -85,B 0,C 180,E1 -12062.352,E2 -12062.352} C_VEL
LIN {X 0,Y 384.396,Z 621.403,A -85,B 0,C 180,E1 -12063.931,E2 -12063.931} C_VEL
LIN {X 0,Y 383.82,Z 627.058,A -85,B 0,C 180,E1 -12065.253,E2 -12065.253} C_VEL
LIN {X 0,Y 383.214,Z 632.556,A -85,B 0,C 180,E1 -12066.846,E2 -12066.846} C_VEL
LIN {X 0,Y 382.757,Z 636.838,A -85,B 0,C 180,E1 -12068.447,E2 -12068.447} C_VEL
LIN {X 0,Y 382.478,Z 639.091,A -85,B 0,C 180,E1 -12069.519,E2 -12069.519} C_VEL
LIN {X 0,Y 382.254,Z 640.876,A -85,B 0,C 180,E1 -12070.594,E2 -12070.594} C_VEL
LIN {X 0,Y 382.097,Z 642.178,A -85,B 0,C 180,E1 -12071.673,E2 -12071.673} C_VEL
LIN {X 0,Y 381.976,Z 643.091,A -85,B 0,C 180,E1 -12072.798,E2 -12072.798} C_VEL
LIN {X 0,Y 381.851,Z 643.514,A -85,B 0,C 180,E1 -12073.843,E2 -12073.843} C_VEL
LIN {X 0,Y 381.818,Z 643.481,A -85,B 0,C 180,E1 -12074.933,E2 -12074.933} C_VEL
LIN {X 0,Y 381.86,Z 642.376,A -85,B 0,C 180,E1 -12076.853,E2 -12076.853} C_VEL
LIN {X 0,Y 381.938,Z 640.719,A -85,B 0,C 180,E1 -12078.229,E2 -12078.229} C_VEL
LIN {X 0,Y 382.106,Z 637.888,A -85,B 0,C 180,E1 -12079.815,E2 -12079.815} C_VEL
LIN {X 0,Y 382.33,Z 633.523,A -85,B 0,C 180,E1 -12081.57,E2 -12081.57} C_VEL
LIN {X 0,Y 382.735,Z 627.652,A -85,B 0,C 180,E1 -12083.345,E2 -12083.345} C_VEL
LIN {X 0,Y 383.208,Z 620.828,A -85,B 0,C 180,E1 -12084.949,E2 -12084.949} C_VEL
LIN {X 0,Y 383.762,Z 613.576,A -85,B 0,C 180,E1 -12086.336,E2 -12086.336} C_VEL
LIN {X 0,Y 384.455,Z 604.316,A -85,B 0,C 180,E1 -12087.785,E2 -12087.785} C_VEL
LIN {X 0,Y 385.061,Z 594.315,A -85,B 0,C 180,E1 -12089.055,E2 -12089.055} C_VEL
LIN {X 0,Y 385.862,Z 582.921,A -85,B 0,C 180,E1 -12090.209,E2 -12090.209} C_VEL
LIN {X 0,Y 386.545,Z 570.526,A -85,B 0,C 180,E1 -12091.2,E2 -12091.2} C_VEL
LIN {X 0,Y 387.161,Z 557.196,A -85,B 0,C 180,E1 -12091.994,E2 -12091.994} C_VEL
LIN {X 0,Y 387.557,Z 544.039,A -85,B 0,C 180,E1 -12092.553,E2 -12092.553} C_VEL
LIN {X 0,Y 387.883,Z 526.783,A -85,B 0,C 180,E1 -12092.988,E2 -12092.988} C_VEL
LIN {X 0,Y 389.241,Z 453.624,A -85,B 0,C 180,E1 -12094.59,E2 -12094.59} C_VEL
LIN {X 0,Y 383.071,Z 435.766,A -85,B 0,C 180,E1 -12095.296,E2 -12095.296} C_VEL
LIN {X 0,Y 382.983,Z 435.779,A -85,B 0,C 180,E1 -12098.603,E2 -12098.603} C_VEL
LIN {X 0,Y 382.963,Z 435.777,A -85,B 0,C 180,E1 -12101.35,E2 -12101.35} C_VEL
LIN {X 0,Y 382.996,Z 435.779,A -85,B 0,C 180,E1 -12104.303,E2 -12104.303} C_VEL
LIN {X 0,Y 383.013,Z 435.771,A -85,B 0,C 180,E1 -12107.24,E2 -12107.24} C_VEL
LIN {X 0,Y 382.987,Z 435.782,A -85,B 0,C 180,E1 -12110.419,E2 -12110.419} C_VEL
LIN {X 0,Y 383.025,Z 435.773,A -85,B 0,C 180,E1 -12114.044,E2 -12114.044} C_VEL
LIN {X 0,Y 382.989,Z 435.774,A -85,B 0,C 180,E1 -12117.578,E2 -12117.578} C_VEL
LIN {X 0,Y 382.98,Z 435.781,A -85,B 0,C 180,E1 -12120.299,E2 -12120.299} C_VEL
LIN {X 0,Y 383.005,Z 435.775,A -85,B 0,C 180,E1 -12124.044,E2 -12124.044} C_VEL
LIN {X 0,Y 382.999,Z 435.773,A -85,B 0,C 180,E1 -12127.334,E2 -12127.334} C_VEL
LIN {X 0,Y 383.06,Z 435.769,A -85,B 0,C 180,E1 -12130.716,E2 -12130.716} C_VEL
LIN {X 0,Y 383.08,Z 435.765,A -85,B 0,C 180,E1 -12134.026,E2 -12134.026} C_VEL
LIN {X 0,Y 383.138,Z 435.756,A -85,B 0,C 180,E1 -12137.284,E2 -12137.284} C_VEL
LIN {X 0,Y 383.145,Z 435.762,A -85,B 0,C 180,E1 -12140.497,E2 -12140.497} C_VEL
LIN {X 0,Y 383.244,Z 435.743,A -85,B 0,C 180,E1 -12143.683,E2 -12143.683} C_VEL
LIN {X 0,Y 383.384,Z 435.726,A -85,B 0,C 180,E1 -12147.899,E2 -12147.899} C_VEL
LIN {X 0,Y 383.513,Z 435.711,A -85,B 0,C 180,E1 -12150,E2 -12150} C_VEL
LIN {X 0,Y 383.212,Z 435.747,A -85,B 0,C 180,E1 -12153.154,E2 -12153.154} C_VEL
LIN {X 0,Y 383.275,Z 435.743,A -85,B 0,C 180,E1 -12156.316,E2 -12156.316} C_VEL
LIN {X 0,Y 383.144,Z 435.755,A -85,B 0,C 180,E1 -12159.502,E2 -12159.502} C_VEL
LIN {X 0,Y 383.126,Z 435.757,A -85,B 0,C 180,E1 -12163.536,E2 -12163.536} C_VEL
LIN {X 0,Y 383.085,Z 435.763,A -85,B 0,C 180,E1 -12166.933,E2 -12166.933} C_VEL
LIN {X 0,Y 382.449,Z 435.846,A -85,B 0,C 180,E1 -12167.811,E2 -12167.811} C_VEL
LIN {X 0,Y 379.559,Z 436.206,A -85,B 0,C 180,E1 -12169.236,E2 -12169.236} C_VEL
LIN {X 0,Y 377.089,Z 436.515,A -85,B 0,C 180,E1 -12170.388,E2 -12170.388} C_VEL
LIN {X 0,Y 376.031,Z 436.642,A -85,B 0,C 180,E1 -12171.28,E2 -12171.28} C_VEL
LIN {X 0,Y 375.948,Z 436.651,A -85,B 0,C 180,E1 -12171.582,E2 -12171.582} C_VEL
LIN {X 0,Y 375.978,Z 436.652,A -85,B 0,C 180,E1 -12174.282,E2 -12174.282} C_VEL
LIN {X 0,Y 375.935,Z 436.654,A -85,B 0,C 180,E1 -12177.863,E2 -12177.863} C_VEL
LIN {X 0,Y 375.957,Z 436.65,A -85,B 0,C 180,E1 -12181.562,E2 -12181.562} C_VEL
LIN {X 0,Y 375.957,Z 436.65,A -85,B 0,C 180,E1 -12185.415,E2 -12185.415} C_VEL
LIN {X 0,Y 375.936,Z 436.656,A -85,B 0,C 180,E1 -12188.263,E2 -12188.263} C_VEL
LIN {X 0,Y 375.919,Z 436.655,A -85,B 0,C 180,E1 -12191.598,E2 -12191.598} C_VEL
LIN {X 0,Y 375.925,Z 436.659,A -85,B 0,C 180,E1 -12194.731,E2 -12194.731} C_VEL
LIN {X 0,Y 375.923,Z 436.659,A -85,B 0,C 180,E1 -12198.401,E2 -12198.401} C_VEL
LIN {X 0,Y 375.961,Z 436.65,A -85,B 0,C 180,E1 -12201.911,E2 -12201.911} C_VEL
LIN {X 0,Y 375.979,Z 436.648,A -85,B 0,C 180,E1 -12205.333,E2 -12205.333} C_VEL
LIN {X 0,Y 375.957,Z 436.655,A -85,B 0,C 180,E1 -12208.438,E2 -12208.438} C_VEL
LIN {X 0,Y 375.982,Z 436.649,A -85,B 0,C 180,E1 -12212.14,E2 -12212.14} C_VEL
LIN {X 0,Y 376.004,Z 436.651,A -85,B 0,C 180,E1 -12214.539,E2 -12214.539} C_VEL
LIN {X 0,Y 375.967,Z 436.65,A -85,B 0,C 180,E1 -12218.046,E2 -12218.046} C_VEL
LIN {X 0,Y 376.006,Z 436.644,A -85,B 0,C 180,E1 -12221.473,E2 -12221.473} C_VEL
LIN {X 0,Y 376.058,Z 436.642,A -85,B 0,C 180,E1 -12224.833,E2 -12224.833} C_VEL
LIN {X 0,Y 376.049,Z 436.641,A -85,B 0,C 180,E1 -12228.137,E2 -12228.137} C_VEL
LIN {X 0,Y 376.213,Z 436.619,A -85,B 0,C 180,E1 -12231.924,E2 -12231.924} C_VEL
LIN {X 0,Y 376.16,Z 436.632,A -85,B 0,C 180,E1 -12234.64,E2 -12234.64} C_VEL
LIN {X 0,Y 376.351,Z 436.601,A -85,B 0,C 180,E1 -12237.86,E2 -12237.86} C_VEL
LIN {X 0,Y 376.487,Z 436.585,A -85,B 0,C 180,E1 -12240,E2 -12240} C_VEL
LIN {X 0,Y 376.186,Z 436.623,A -85,B 0,C 180,E1 -12243.213,E2 -12243.213} C_VEL
LIN {X 0,Y 376.246,Z 436.618,A -85,B 0,C 180,E1 -12246.435,E2 -12246.435} C_VEL
LIN {X 0,Y 376.205,Z 436.625,A -85,B 0,C 180,E1 -12248.595,E2 -12248.595} C_VEL
LIN {X 0,Y 376.049,Z 436.639,A -85,B 0,C 180,E1 -12251.864,E2 -12251.864} C_VEL
LIN {X 0,Y 376.058,Z 436.639,A -85,B 0,C 180,E1 -12255.168,E2 -12255.168} C_VEL
LIN {X 0,Y 376.023,Z 436.647,A -85,B 0,C 180,E1 -12258.526,E2 -12258.526} C_VEL
LIN {X 0,Y 375.956,Z 436.651,A -85,B 0,C 180,E1 -12261.955,E2 -12261.955} C_VEL
LIN {X 0,Y 376.004,Z 436.645,A -85,B 0,C 180,E1 -12265.461,E2 -12265.461} C_VEL
LIN {X 0,Y 375.97,Z 436.651,A -85,B 0,C 180,E1 -12269.079,E2 -12269.079} C_VEL
LIN {X 0,Y 375.949,Z 436.657,A -85,B 0,C 180,E1 -12272.829,E2 -12272.829} C_VEL
LIN {X 0,Y 375.957,Z 436.651,A -85,B 0,C 180,E1 -12275.416,E2 -12275.416} C_VEL
LIN {X 0,Y 375.973,Z 436.65,A -85,B 0,C 180,E1 -12278.271,E2 -12278.271} C_VEL
LIN {X 0,Y 375.934,Z 436.653,A -85,B 0,C 180,E1 -12281.601,E2 -12281.601} C_VEL
LIN {X 0,Y 375.928,Z 436.655,A -85,B 0,C 180,E1 -12285.269,E2 -12285.269} C_VEL
LIN {X 0,Y 375.936,Z 436.656,A -85,B 0,C 180,E1 -12288.399,E2 -12288.399} C_VEL
LIN {X 0,Y 375.974,Z 436.648,A -85,B 0,C 180,E1 -12291.73,E2 -12291.73} C_VEL
LIN {X 0,Y 375.98,Z 436.651,A -85,B 0,C 180,E1 -12295.333,E2 -12295.333} C_VEL
LIN {X 0,Y 375.987,Z 436.739,A -85,B 0,C 180,E1 -12298.838,E2 -12298.838} C_VEL
LIN {X 0,Y 379.213,Z 451.627,A -85,B 0,C 180,E1 -12302.098,E2 -12302.098} C_VEL
LIN {X 0,Y 380.211,Z 457.751,A -85,B 0,C 180,E1 -12303.386,E2 -12303.386} C_VEL
LIN {X 0,Y 378.739,Z 475.099,A -85,B 0,C 180,E1 -12306.777,E2 -12306.777} C_VEL
LIN {X 0,Y 377.815,Z 488.496,A -85,B 0,C 180,E1 -12309.357,E2 -12309.357} C_VEL
LIN {X 0,Y 381.946,Z 524.147,A -85,B 0,C 180,E1 -12310.379,E2 -12310.379} C_VEL
LIN {X 0,Y 380.43,Z 598.787,A -85,B 0,C 180,E1 -12312.079,E2 -12312.079} C_VEL
LIN {X 0,Y 379.806,Z 611.616,A -85,B 0,C 180,E1 -12312.571,E2 -12312.571} C_VEL
LIN {X 0,Y 378.999,Z 624.698,A -85,B 0,C 180,E1 -12313.296,E2 -12313.296} C_VEL
LIN {X 0,Y 378.216,Z 637.114,A -85,B 0,C 180,E1 -12314.231,E2 -12314.231} C_VEL
LIN {X 0,Y 377.336,Z 648.656,A -85,B 0,C 180,E1 -12315.341,E2 -12315.341} C_VEL
LIN {X 0,Y 376.659,Z 658.391,A -85,B 0,C 180,E1 -12316.513,E2 -12316.513} C_VEL
LIN {X 0,Y 375.968,Z 667.565,A -85,B 0,C 180,E1 -12317.861,E2 -12317.861} C_VEL
LIN {X 0,Y 375.3,Z 676.509,A -85,B 0,C 180,E1 -12319.48,E2 -12319.48} C_VEL
LIN {X 0,Y 374.972,Z 683.626,A -85,B 0,C 180,E1 -12321.105,E2 -12321.105} C_VEL
LIN {X 0,Y 374.751,Z 690.122,A -85,B 0,C 180,E1 -12322.999,E2 -12322.999} C_VEL
LIN {X 0,Y 374.728,Z 694.328,A -85,B 0,C 180,E1 -12324.62,E2 -12324.62} C_VEL
LIN {X 0,Y 374.674,Z 696.48,A -85,B 0,C 180,E1 -12325.697,E2 -12325.697} C_VEL
LIN {X 0,Y 374.791,Z 698.166,A -85,B 0,C 180,E1 -12326.775,E2 -12326.775} C_VEL
LIN {X 0,Y 374.806,Z 699.408,A -85,B 0,C 180,E1 -12327.851,E2 -12327.851} C_VEL
LIN {X 0,Y 374.845,Z 700.205,A -85,B 0,C 180,E1 -12328.926,E2 -12328.926} C_VEL
LIN {X 0,Y 374.864,Z 700.531,A -85,B 0,C 180,E1 -12330,E2 -12330} C_VEL
LIN {X 0,Y 374.792,Z 700.43,A -85,B 0,C 180,E1 -12331.075,E2 -12331.075} C_VEL
LIN {X 0,Y 374.794,Z 699.917,A -85,B 0,C 180,E1 -12332.15,E2 -12332.15} C_VEL
LIN {X 0,Y 374.698,Z 698.94,A -85,B 0,C 180,E1 -12333.226,E2 -12333.226} C_VEL
LIN {X 0,Y 374.65,Z 697.517,A -85,B 0,C 180,E1 -12334.304,E2 -12334.304} C_VEL
LIN {X 0,Y 374.621,Z 694.117,A -85,B 0,C 180,E1 -12336.121,E2 -12336.121} C_VEL
LIN {X 0,Y 374.849,Z 688.937,A -85,B 0,C 180,E1 -12338.084,E2 -12338.084} C_VEL
LIN {X 0,Y 375.225,Z 682.234,A -85,B 0,C 180,E1 -12339.977,E2 -12339.977} C_VEL
LIN {X 0,Y 375.811,Z 674.982,A -85,B 0,C 180,E1 -12341.598,E2 -12341.598} C_VEL
LIN {X 0,Y 376.548,Z 665.974,A -85,B 0,C 180,E1 -12343.217,E2 -12343.217} C_VEL
LIN {X 0,Y 377.496,Z 656.558,A -85,B 0,C 180,E1 -12344.586,E2 -12344.586} C_VEL
LIN {X 0,Y 378.626,Z 645.532,A -85,B 0,C 180,E1 -12345.89,E2 -12345.89} C_VEL
LIN {X 0,Y 379.745,Z 634.347,A -85,B 0,C 180,E1 -12346.947,E2 -12346.947} C_VEL
LIN {X 0,Y 380.924,Z 622.024,A -85,B 0,C 180,E1 -12347.863,E2 -12347.863} C_VEL
LIN {X 0,Y 381.812,Z 610.643,A -85,B 0,C 180,E1 -12348.513,E2 -12348.513} C_VEL
LIN {X 0,Y 382.692,Z 597.183,A -85,B 0,C 180,E1 -12349.06,E2 -12349.06} C_VEL
LIN {X 0,Y 383.33,Z 575.223,A -85,B 0,C 180,E1 -12349.618,E2 -12349.618} C_VEL
LIN {X 0,Y 384.786,Z 522.98,A -85,B 0,C 180,E1 -12350.875,E2 -12350.875} C_VEL
LIN {X 0,Y 382.547,Z 503.148,A -85,B 0,C 180,E1 -12351.59,E2 -12351.59} C_VEL
LIN {X 0,Y 379.438,Z 485.811,A -85,B 0,C 180,E1 -12352.326,E2 -12352.326} C_VEL
LIN {X 0,Y 378.95,Z 483.085,A -85,B 0,C 180,E1 -12352.468,E2 -12352.468} C_VEL
LIN {X 0,Y 380.995,Z 464.694,A -85,B 0,C 180,E1 -12356.278,E2 -12356.278} C_VEL
LIN {X 0,Y 381.364,Z 460.697,A -85,B 0,C 180,E1 -12357.137,E2 -12357.137} C_VEL
LIN {X 0,Y 380.091,Z 453.066,A -85,B 0,C 180,E1 -12359.001,E2 -12359.001} C_VEL
LIN {X 0,Y 377.652,Z 442.922,A -85,B 0,C 180,E1 -12361.718,E2 -12361.718} C_VEL
LIN {X 0,Y 375.968,Z 436.661,A -85,B 0,C 180,E1 -12363.587,E2 -12363.587} C_VEL
LIN {X 0,Y 375.957,Z 436.657,A -85,B 0,C 180,E1 -12366.741,E2 -12366.741} C_VEL
LIN {X 0,Y 375.992,Z 436.651,A -85,B 0,C 180,E1 -12369.971,E2 -12369.971} C_VEL
LIN {X 0,Y 375.933,Z 436.656,A -85,B 0,C 180,E1 -12373.766,E2 -12373.766} C_VEL
LIN {X 0,Y 375.938,Z 436.657,A -85,B 0,C 180,E1 -12376.811,E2 -12376.811} C_VEL
LIN {X 0,Y 375.964,Z 436.655,A -85,B 0,C 180,E1 -12380.537,E2 -12380.537} C_VEL
LIN {X 0,Y 375.967,Z 436.649,A -85,B 0,C 180,E1 -12383.496,E2 -12383.496} C_VEL
LIN {X 0,Y 375.964,Z 436.65,A -85,B 0,C 180,E1 -12385.889,E2 -12385.889} C_VEL
LIN {X 0,Y 375.965,Z 436.65,A -85,B 0,C 180,E1 -12389.687,E2 -12389.687} C_VEL
LIN {X 0,Y 375.929,Z 436.656,A -85,B 0,C 180,E1 -12392.136,E2 -12392.136} C_VEL
LIN {X 0,Y 375.94,Z 436.658,A -85,B 0,C 180,E1 -12394.534,E2 -12394.534} C_VEL
LIN {X 0,Y 375.977,Z 436.652,A -85,B 0,C 180,E1 -12396.887,E2 -12396.887} C_VEL
LIN {X 0,Y 375.961,Z 436.656,A -85,B 0,C 180,E1 -12400.337,E2 -12400.337} C_VEL
LIN {X 0,Y 375.956,Z 436.656,A -85,B 0,C 180,E1 -12403.716,E2 -12403.716} C_VEL
LIN {X 0,Y 376.078,Z 436.639,A -85,B 0,C 180,E1 -12407.041,E2 -12407.041} C_VEL
LIN {X 0,Y 376.109,Z 436.637,A -85,B 0,C 180,E1 -12410.318,E2 -12410.318} C_VEL
LIN {X 0,Y 376.145,Z 436.744,A -85,B 0,C 180,E1 -12411.459,E2 -12411.459} C_VEL
LIN {X 0,Y 376.855,Z 439.496,A -85,B 0,C 180,E1 -12412.465,E2 -12412.465} C_VEL
LIN {X 0,Y 383.074,Z 452.387,A -85,B 0,C 180,E1 -12413.396,E2 -12413.396} C_VEL
LIN {X 0,Y 386.392,Z 460.46,A -85,B 0,C 180,E1 -12413.897,E2 -12413.897} C_VEL
LIN {X 0,Y 383.545,Z 544.484,A -85,B 0,C 180,E1 -12415.961,E2 -12415.961} C_VEL
LIN {X 0,Y 383.102,Z 558.018,A -85,B 0,C 180,E1 -12416.516,E2 -12416.516} C_VEL
LIN {X 0,Y 382.48,Z 570.342,A -85,B 0,C 180,E1 -12417.235,E2 -12417.235} C_VEL
LIN {X 0,Y 381.536,Z 582.306,A -85,B 0,C 180,E1 -12418.153,E2 -12418.153} C_VEL
LIN {X 0,Y 380.62,Z 592.952,A -85,B 0,C 180,E1 -12419.192,E2 -12419.192} C_VEL
LIN {X 0,Y 379.53,Z 603.665,A -85,B 0,C 180,E1 -12420.503,E2 -12420.503} C_VEL
LIN {X 0,Y 378.637,Z 612.572,A -85,B 0,C 180,E1 -12421.861,E2 -12421.861} C_VEL
LIN {X 0,Y 377.648,Z 621.149,A -85,B 0,C 180,E1 -12423.467,E2 -12423.467} C_VEL
LIN {X 0,Y 376.879,Z 627.968,A -85,B 0,C 180,E1 -12425.082,E2 -12425.082} C_VEL
LIN {X 0,Y 376.144,Z 634.211,A -85,B 0,C 180,E1 -12426.976,E2 -12426.976} C_VEL
LIN {X 0,Y 375.672,Z 638.251,A -85,B 0,C 180,E1 -12428.607,E2 -12428.607} C_VEL
LIN {X 0,Y 375.396,Z 640.322,A -85,B 0,C 180,E1 -12429.7,E2 -12429.7} C_VEL
LIN {X 0,Y 375.154,Z 641.934,A -85,B 0,C 180,E1 -12430.797,E2 -12430.797} C_VEL
LIN {X 0,Y 375.018,Z 643.114,A -85,B 0,C 180,E1 -12431.896,E2 -12431.896} C_VEL
LIN {X 0,Y 374.89,Z 643.831,A -85,B 0,C 180,E1 -12433.001,E2 -12433.001} C_VEL
LIN {X 0,Y 374.779,Z 644.104,A -85,B 0,C 180,E1 -12434.11,E2 -12434.11} C_VEL
LIN {X 0,Y 374.74,Z 643.954,A -85,B 0,C 180,E1 -12435.222,E2 -12435.222} C_VEL
LIN {X 0,Y 374.784,Z 642.779,A -85,B 0,C 180,E1 -12436.987,E2 -12436.987} C_VEL
LIN {X 0,Y 374.961,Z 639.741,A -85,B 0,C 180,E1 -12439.148,E2 -12439.148} C_VEL
LIN {X 0,Y 375.168,Z 636.083,A -85,B 0,C 180,E1 -12440.85,E2 -12440.85} C_VEL
LIN {X 0,Y 375.466,Z 631.149,A -85,B 0,C 180,E1 -12442.564,E2 -12442.564} C_VEL
LIN {X 0,Y 375.921,Z 624.72,A -85,B 0,C 180,E1 -12444.286,E2 -12444.286} C_VEL
LIN {X 0,Y 376.607,Z 616.593,A -85,B 0,C 180,E1 -12446,E2 -12446} C_VEL
LIN {X 0,Y 377.18,Z 608.021,A -85,B 0,C 180,E1 -12447.462,E2 -12447.462} C_VEL
LIN {X 0,Y 377.878,Z 598.586,A -85,B 0,C 180,E1 -12448.766,E2 -12448.766} C_VEL
LIN {X 0,Y 378.58,Z 588.193,A -85,B 0,C 180,E1 -12449.938,E2 -12449.938} C_VEL
LIN {X 0,Y 379.271,Z 577.117,A -85,B 0,C 180,E1 -12450.945,E2 -12450.945} C_VEL
LIN {X 0,Y 379.874,Z 565.76,A -85,B 0,C 180,E1 -12451.758,E2 -12451.758} C_VEL
LIN {X 0,Y 380.423,Z 552.323,A -85,B 0,C 180,E1 -12452.473,E2 -12452.473} C_VEL
LIN {X 0,Y 380.822,Z 539.378,A -85,B 0,C 180,E1 -12452.945,E2 -12452.945} C_VEL
LIN {X 0,Y 382.432,Z 455.036,A -85,B 0,C 180,E1 -12454.849,E2 -12454.849} C_VEL
LIN {X 0,Y 376.006,Z 436.646,A -85,B 0,C 180,E1 -12455.583,E2 -12455.583} C_VEL
LIN {X 0,Y 375.936,Z 436.653,A -85,B 0,C 180,E1 -12459.466,E2 -12459.466} C_VEL
LIN {X 0,Y 375.936,Z 436.653,A -85,B 0,C 180,E1 -12463.189,E2 -12463.189} C_VEL
LIN {X 0,Y 375.936,Z 436.655,A -85,B 0,C 180,E1 -12466.81,E2 -12466.81} C_VEL
LIN {X 0,Y 375.935,Z 436.658,A -85,B 0,C 180,E1 -12470.533,E2 -12470.533} C_VEL
LIN {X 0,Y 375.964,Z 436.649,A -85,B 0,C 180,E1 -12473.496,E2 -12473.496} C_VEL
LIN {X 0,Y 375.962,Z 436.651,A -85,B 0,C 180,E1 -12475.888,E2 -12475.888} C_VEL
LIN {X 0,Y 375.964,Z 436.65,A -85,B 0,C 180,E1 -12479.687,E2 -12479.687} C_VEL
LIN {X 0,Y 375.929,Z 436.657,A -85,B 0,C 180,E1 -12482.135,E2 -12482.135} C_VEL
LIN {X 0,Y 375.975,Z 436.649,A -85,B 0,C 180,E1 -12485.717,E2 -12485.717} C_VEL
LIN {X 0,Y 376,Z 436.645,A -85,B 0,C 180,E1 -12489.198,E2 -12489.198} C_VEL
LIN {X 0,Y 376.052,Z 436.644,A -85,B 0,C 180,E1 -12492.601,E2 -12492.601} C_VEL
LIN {X 0,Y 376.091,Z 436.639,A -85,B 0,C 180,E1 -12496.342,E2 -12496.342} C_VEL
LIN {X 0,Y 376.115,Z 436.636,A -85,B 0,C 180,E1 -12500.318,E2 -12500.318} C_VEL
LIN {X 0,Y 376.202,Z 436.62,A -85,B 0,C 180,E1 -12503.564,E2 -12503.564} C_VEL
LIN {X 0,Y 376.35,Z 436.602,A -85,B 0,C 180,E1 -12507.859,E2 -12507.859} C_VEL
LIN {X 0,Y 376.483,Z 436.587,A -85,B 0,C 180,E1 -12510,E2 -12510} C_VEL
LIN {X 0,Y 376.344,Z 436.605,A -85,B 0,C 180,E1 -12512.14,E2 -12512.14} C_VEL
LIN {X 0,Y 376.231,Z 436.622,A -85,B 0,C 180,E1 -12516.435,E2 -12516.435} C_VEL
LIN {X 0,Y 376.114,Z 436.631,A -85,B 0,C 180,E1 -12519.681,E2 -12519.681} C_VEL
LIN {X 0,Y 376.09,Z 436.634,A -85,B 0,C 180,E1 -12523.657,E2 -12523.657} C_VEL
LIN {X 0,Y 376.033,Z 436.641,A -85,B 0,C 180,E1 -12527.399,E2 -12527.399} C_VEL
LIN {X 0,Y 375.979,Z 436.651,A -85,B 0,C 180,E1 -12530.832,E2 -12530.832} C_VEL
LIN {X 0,Y 375.948,Z 436.651,A -85,B 0,C 180,E1 -12531.582,E2 -12531.582} C_VEL
LIN {X 0,Y 375.299,Z 436.739,A -85,B 0,C 180,E1 -12532.476,E2 -12532.476} C_VEL
LIN {X 0,Y 372.481,Z 437.084,A -85,B 0,C 180,E1 -12533.932,E2 -12533.932} C_VEL
LIN {X 0,Y 370.072,Z 437.385,A -85,B 0,C 180,E1 -12535.108,E2 -12535.108} C_VEL
LIN {X 0,Y 369.013,Z 437.517,A -85,B 0,C 180,E1 -12536.017,E2 -12536.017} C_VEL
LIN {X 0,Y 368.914,Z 437.532,A -85,B 0,C 180,E1 -12536.326,E2 -12536.326} C_VEL
LIN {X 0,Y 368.896,Z 437.53,A -85,B 0,C 180,E1 -12539.692,E2 -12539.692} C_VEL
LIN {X 0,Y 368.897,Z 437.532,A -85,B 0,C 180,E1 -12543.043,E2 -12543.043} C_VEL
LIN {X 0,Y 368.916,Z 437.53,A -85,B 0,C 180,E1 -12546.197,E2 -12546.197} C_VEL
LIN {X 0,Y 368.874,Z 437.535,A -85,B 0,C 180,E1 -12548.956,E2 -12548.956} C_VEL
LIN {X 0,Y 368.871,Z 437.534,A -85,B 0,C 180,E1 -12552.007,E2 -12552.007} C_VEL
LIN {X 0,Y 368.878,Z 437.533,A -85,B 0,C 180,E1 -12555.175,E2 -12555.175} C_VEL
LIN {X 0,Y 368.873,Z 437.535,A -85,B 0,C 180,E1 -12558.176,E2 -12558.176} C_VEL
LIN {X 0,Y 368.904,Z 437.529,A -85,B 0,C 180,E1 -12561.36,E2 -12561.36} C_VEL
LIN {X 0,Y 368.935,Z 437.526,A -85,B 0,C 180,E1 -12565.146,E2 -12565.146} C_VEL
LIN {X 0,Y 368.928,Z 437.528,A -85,B 0,C 180,E1 -12569.046,E2 -12569.046} C_VEL
LIN {X 0,Y 368.962,Z 437.526,A -85,B 0,C 180,E1 -12572.796,E2 -12572.796} C_VEL
LIN {X 0,Y 368.943,Z 437.526,A -85,B 0,C 180,E1 -12576.113,E2 -12576.113} C_VEL
LIN {X 0,Y 368.935,Z 437.526,A -85,B 0,C 180,E1 -12579.947,E2 -12579.947} C_VEL
LIN {X 0,Y 368.975,Z 437.52,A -85,B 0,C 180,E1 -12583.399,E2 -12583.399} C_VEL
LIN {X 0,Y 369.057,Z 437.515,A -85,B 0,C 180,E1 -12586.79,E2 -12586.79} C_VEL
LIN {X 0,Y 369.066,Z 437.51,A -85,B 0,C 180,E1 -12590.132,E2 -12590.132} C_VEL
LIN {X 0,Y 369.152,Z 437.501,A -85,B 0,C 180,E1 -12592.342,E2 -12592.342} C_VEL
LIN {X 0,Y 369.132,Z 437.506,A -85,B 0,C 180,E1 -12594.537,E2 -12594.537} C_VEL
LIN {X 0,Y 369.316,Z 437.478,A -85,B 0,C 180,E1 -12597.819,E2 -12597.819} C_VEL
LIN {X 0,Y 369.456,Z 437.461,A -85,B 0,C 180,E1 -12600,E2 -12600} C_VEL
LIN {X 0,Y 369.317,Z 437.479,A -85,B 0,C 180,E1 -12602.181,E2 -12602.181} C_VEL
LIN {X 0,Y 369.208,Z 437.497,A -85,B 0,C 180,E1 -12606.558,E2 -12606.558} C_VEL
LIN {X 0,Y 369.137,Z 437.506,A -85,B 0,C 180,E1 -12608.761,E2 -12608.761} C_VEL
LIN {X 0,Y 369.004,Z 437.518,A -85,B 0,C 180,E1 -12612.093,E2 -12612.093} C_VEL
LIN {X 0,Y 368.998,Z 437.517,A -85,B 0,C 180,E1 -12615.465,E2 -12615.465} C_VEL
LIN {X 0,Y 368.982,Z 437.524,A -85,B 0,C 180,E1 -12618.893,E2 -12618.893} C_VEL
LIN {X 0,Y 368.922,Z 437.53,A -85,B 0,C 180,E1 -12622.396,E2 -12622.396} C_VEL
LIN {X 0,Y 368.999,Z 437.518,A -85,B 0,C 180,E1 -12625.98,E2 -12625.98} C_VEL
LIN {X 0,Y 368.961,Z 437.527,A -85,B 0,C 180,E1 -12628.812,E2 -12628.812} C_VEL
LIN {X 0,Y 368.898,Z 437.532,A -85,B 0,C 180,E1 -12632.238,E2 -12632.238} C_VEL
LIN {X 0,Y 368.928,Z 437.529,A -85,B 0,C 180,E1 -12635.002,E2 -12635.002} C_VEL
LIN {X 0,Y 368.908,Z 437.534,A -85,B 0,C 180,E1 -12638.641,E2 -12638.641} C_VEL
LIN {X 0,Y 368.881,Z 437.532,A -85,B 0,C 180,E1 -12642.01,E2 -12642.01} C_VEL
LIN {X 0,Y 368.886,Z 437.533,A -85,B 0,C 180,E1 -12645.177,E2 -12645.177} C_VEL
LIN {X 0,Y 368.884,Z 437.533,A -85,B 0,C 180,E1 -12648.178,E2 -12648.178} C_VEL
LIN {X 0,Y 368.909,Z 437.529,A -85,B 0,C 180,E1 -12651.36,E2 -12651.36} C_VEL
LIN {X 0,Y 368.937,Z 437.53,A -85,B 0,C 180,E1 -12655.147,E2 -12655.147} C_VEL
LIN {X 0,Y 368.933,Z 437.579,A -85,B 0,C 180,E1 -12658.569,E2 -12658.569} C_VEL
LIN {X 0,Y 372.06,Z 452.15,A -85,B 0,C 180,E1 -12661.821,E2 -12661.821} C_VEL
LIN {X 0,Y 373.203,Z 458.214,A -85,B 0,C 180,E1 -12663.131,E2 -12663.131} C_VEL
LIN {X 0,Y 372.294,Z 469.838,A -85,B 0,C 180,E1 -12665.462,E2 -12665.462} C_VEL
LIN {X 0,Y 370.821,Z 488.004,A -85,B 0,C 180,E1 -12669.041,E2 -12669.041} C_VEL
LIN {X 0,Y 375.064,Z 525.206,A -85,B 0,C 180,E1 -12670.132,E2 -12670.132} C_VEL
LIN {X 0,Y 373.521,Z 598.443,A -85,B 0,C 180,E1 -12671.843,E2 -12671.843} C_VEL
LIN {X 0,Y 372.84,Z 611.909,A -85,B 0,C 180,E1 -12672.376,E2 -12672.376} C_VEL
LIN {X 0,Y 372.017,Z 624.721,A -85,B 0,C 180,E1 -12673.115,E2 -12673.115} C_VEL
LIN {X 0,Y 371.294,Z 635.435,A -85,B 0,C 180,E1 -12673.929,E2 -12673.929} C_VEL
LIN {X 0,Y 370.474,Z 646.838,A -85,B 0,C 180,E1 -12675.021,E2 -12675.021} C_VEL
LIN {X 0,Y 369.665,Z 657.333,A -85,B 0,C 180,E1 -12676.279,E2 -12676.279} C_VEL
LIN {X 0,Y 368.94,Z 666.439,A -85,B 0,C 180,E1 -12677.626,E2 -12677.626} C_VEL
LIN {X 0,Y 368.277,Z 675.505,A -85,B 0,C 180,E1 -12679.277,E2 -12679.277} C_VEL
LIN {X 0,Y 367.907,Z 682.735,A -85,B 0,C 180,E1 -12680.933,E2 -12680.933} C_VEL
LIN {X 0,Y 367.737,Z 687.637,A -85,B 0,C 180,E1 -12682.312,E2 -12682.312} C_VEL
LIN {X 0,Y 367.663,Z 691.677,A -85,B 0,C 180,E1 -12683.721,E2 -12683.721} C_VEL
LIN {X 0,Y 367.607,Z 695.792,A -85,B 0,C 180,E1 -12685.615,E2 -12685.615} C_VEL
LIN {X 0,Y 367.698,Z 697.503,A -85,B 0,C 180,E1 -12686.713,E2 -12686.713} C_VEL
LIN {X 0,Y 367.74,Z 698.772,A -85,B 0,C 180,E1 -12687.81,E2 -12687.81} C_VEL
LIN {X 0,Y 367.768,Z 699.608,A -85,B 0,C 180,E1 -12688.905,E2 -12688.905} C_VEL
LIN {X 0,Y 367.798,Z 699.965,A -85,B 0,C 180,E1 -12690,E2 -12690} C_VEL
LIN {X 0,Y 367.719,Z 699.882,A -85,B 0,C 180,E1 -12691.096,E2 -12691.096} C_VEL
LIN {X 0,Y 367.724,Z 699.389,A -85,B 0,C 180,E1 -12692.191,E2 -12692.191} C_VEL
LIN {X 0,Y 367.602,Z 698.451,A -85,B 0,C 180,E1 -12693.288,E2 -12693.288} C_VEL
LIN {X 0,Y 367.574,Z 697.051,A -85,B 0,C 180,E1 -12694.387,E2 -12694.387} C_VEL
LIN {X 0,Y 367.527,Z 694.035,A -85,B 0,C 180,E1 -12696.083,E2 -12696.083} C_VEL
LIN {X 0,Y 367.697,Z 690.146,A -85,B 0,C 180,E1 -12697.689,E2 -12697.689} C_VEL
LIN {X 0,Y 367.951,Z 684.987,A -85,B 0,C 180,E1 -12699.344,E2 -12699.344} C_VEL
LIN {X 0,Y 368.415,Z 678.511,A -85,B 0,C 180,E1 -12700.998,E2 -12700.998} C_VEL
LIN {X 0,Y 369.191,Z 670.509,A -85,B 0,C 180,E1 -12702.646,E2 -12702.646} C_VEL
LIN {X 0,Y 370.045,Z 662.417,A -85,B 0,C 180,E1 -12704.014,E2 -12704.014} C_VEL
LIN {X 0,Y 371.043,Z 652.606,A -85,B 0,C 180,E1 -12705.378,E2 -12705.378} C_VEL
LIN {X 0,Y 372.226,Z 641.824,A -85,B 0,C 180,E1 -12706.594,E2 -12706.594} C_VEL
LIN {X 0,Y 373.485,Z 629.932,A -85,B 0,C 180,E1 -12707.664,E2 -12707.664} C_VEL
LIN {X 0,Y 374.667,Z 616.38,A -85,B 0,C 180,E1 -12708.596,E2 -12708.596} C_VEL
LIN {X 0,Y 375.828,Z 603.24,A -85,B 0,C 180,E1 -12709.244,E2 -12709.244} C_VEL
LIN {X 0,Y 376.509,Z 588.266,A -85,B 0,C 180,E1 -12709.74,E2 -12709.74} C_VEL
LIN {X 0,Y 378.46,Z 524.42,A -85,B 0,C 180,E1 -12711.317,E2 -12711.317} C_VEL
LIN {X 0,Y 376.423,Z 505.316,A -85,B 0,C 180,E1 -12712.018,E2 -12712.018} C_VEL
LIN {X 0,Y 373.478,Z 488.278,A -85,B 0,C 180,E1 -12712.769,E2 -12712.769} C_VEL
LIN {X 0,Y 372.269,Z 482.4,A -85,B 0,C 180,E1 -12713.063,E2 -12713.063} C_VEL
LIN {X 0,Y 374.372,Z 464.939,A -85,B 0,C 180,E1 -12716.779,E2 -12716.779} C_VEL
LIN {X 0,Y 374.596,Z 462.305,A -85,B 0,C 180,E1 -12717.366,E2 -12717.366} C_VEL
LIN {X 0,Y 373.049,Z 453.468,A -85,B 0,C 180,E1 -12719.607,E2 -12719.607} C_VEL
LIN {X 0,Y 370.589,Z 443.71,A -85,B 0,C 180,E1 -12722.355,E2 -12722.355} C_VEL
LIN {X 0,Y 368.939,Z 437.536,A -85,B 0,C 180,E1 -12724.274,E2 -12724.274} C_VEL
LIN {X 0,Y 368.907,Z 437.534,A -85,B 0,C 180,E1 -12727.563,E2 -12727.563} C_VEL
LIN {X 0,Y 368.914,Z 437.533,A -85,B 0,C 180,E1 -12730.37,E2 -12730.37} C_VEL
LIN {X 0,Y 368.886,Z 437.534,A -85,B 0,C 180,E1 -12733.616,E2 -12733.616} C_VEL
LIN {X 0,Y 368.889,Z 437.536,A -85,B 0,C 180,E1 -12736.696,E2 -12736.696} C_VEL
LIN {X 0,Y 368.914,Z 437.53,A -85,B 0,C 180,E1 -12739.643,E2 -12739.643} C_VEL
LIN {X 0,Y 368.904,Z 437.53,A -85,B 0,C 180,E1 -12743.145,E2 -12743.145} C_VEL
LIN {X 0,Y 368.9,Z 437.535,A -85,B 0,C 180,E1 -12746.462,E2 -12746.462} C_VEL
LIN {X 0,Y 368.933,Z 437.527,A -85,B 0,C 180,E1 -12749.047,E2 -12749.047} C_VEL
LIN {X 0,Y 368.868,Z 437.538,A -85,B 0,C 180,E1 -12752.789,E2 -12752.789} C_VEL
LIN {X 0,Y 368.949,Z 437.528,A -85,B 0,C 180,E1 -12756.42,E2 -12756.42} C_VEL
LIN {X 0,Y 368.899,Z 437.533,A -85,B 0,C 180,E1 -12759.945,E2 -12759.945} C_VEL
LIN {X 0,Y 368.904,Z 437.533,A -85,B 0,C 180,E1 -12763.395,E2 -12763.395} C_VEL
LIN {X 0,Y 369.026,Z 437.518,A -85,B 0,C 180,E1 -12766.789,E2 -12766.789} C_VEL
LIN {X 0,Y 369.09,Z 437.577,A -85,B 0,C 180,E1 -12770.755,E2 -12770.755} C_VEL
LIN {X 0,Y 369.853,Z 440.43,A -85,B 0,C 180,E1 -12771.822,E2 -12771.822} C_VEL
LIN {X 0,Y 376.534,Z 453.678,A -85,B 0,C 180,E1 -12772.858,E2 -12772.858} C_VEL
LIN {X 0,Y 380.078,Z 462.293,A -85,B 0,C 180,E1 -12773.43,E2 -12773.43} C_VEL
LIN {X 0,Y 377.117,Z 545.267,A -85,B 0,C 180,E1 -12775.524,E2 -12775.524} C_VEL
LIN {X 0,Y 376.61,Z 559.285,A -85,B 0,C 180,E1 -12776.121,E2 -12776.121} C_VEL
LIN {X 0,Y 375.981,Z 570.415,A -85,B 0,C 180,E1 -12776.785,E2 -12776.785} C_VEL
LIN {X 0,Y 375.007,Z 582.429,A -85,B 0,C 180,E1 -12777.718,E2 -12777.718} C_VEL
LIN {X 0,Y 374.028,Z 593.308,A -85,B 0,C 180,E1 -12778.789,E2 -12778.789} C_VEL
LIN {X 0,Y 372.971,Z 603.234,A -85,B 0,C 180,E1 -12780,E2 -12780} C_VEL
LIN {X 0,Y 372.047,Z 612.148,A -85,B 0,C 180,E1 -12781.353,E2 -12781.353} C_VEL
LIN {X 0,Y 370.934,Z 620.912,A -85,B 0,C 180,E1 -12782.987,E2 -12782.987} C_VEL
LIN {X 0,Y 370.06,Z 627.918,A -85,B 0,C 180,E1 -12784.63,E2 -12784.63} C_VEL
LIN {X 0,Y 369.272,Z 634.263,A -85,B 0,C 180,E1 -12786.557,E2 -12786.557} C_VEL
LIN {X 0,Y 368.741,Z 638.431,A -85,B 0,C 180,E1 -12788.218,E2 -12788.218} C_VEL
LIN {X 0,Y 368.29,Z 641.501,A -85,B 0,C 180,E1 -12789.889,E2 -12789.889} C_VEL
LIN {X 0,Y 368.06,Z 642.987,A -85,B 0,C 180,E1 -12791.008,E2 -12791.008} C_VEL
LIN {X 0,Y 367.833,Z 644.448,A -85,B 0,C 180,E1 -12792.982,E2 -12792.982} C_VEL
LIN {X 0,Y 367.699,Z 644.695,A -85,B 0,C 180,E1 -12794.387,E2 -12794.387} C_VEL
LIN {X 0,Y 367.657,Z 644.355,A -85,B 0,C 180,E1 -12795.523,E2 -12795.523} C_VEL
LIN {X 0,Y 367.703,Z 643.139,A -85,B 0,C 180,E1 -12797.124,E2 -12797.124} C_VEL
LIN {X 0,Y 367.848,Z 640.611,A -85,B 0,C 180,E1 -12798.953,E2 -12798.953} C_VEL
LIN {X 0,Y 368.044,Z 637.129,A -85,B 0,C 180,E1 -12800.66,E2 -12800.66} C_VEL
LIN {X 0,Y 368.349,Z 632.251,A -85,B 0,C 180,E1 -12802.432,E2 -12802.432} C_VEL
LIN {X 0,Y 368.825,Z 626.049,A -85,B 0,C 180,E1 -12804.175,E2 -12804.175} C_VEL
LIN {X 0,Y 369.478,Z 617.994,A -85,B 0,C 180,E1 -12805.944,E2 -12805.944} C_VEL
LIN {X 0,Y 370.079,Z 609.669,A -85,B 0,C 180,E1 -12807.421,E2 -12807.421} C_VEL
LIN {X 0,Y 370.834,Z 600.556,A -85,B 0,C 180,E1 -12808.744,E2 -12808.744} C_VEL
LIN {X 0,Y 371.503,Z 590.557,A -85,B 0,C 180,E1 -12809.931,E2 -12809.931} C_VEL
LIN {X 0,Y 372.306,Z 578.036,A -85,B 0,C 180,E1 -12811.115,E2 -12811.115} C_VEL
LIN {X 0,Y 372.978,Z 565.715,A -85,B 0,C 180,E1 -12812.011,E2 -12812.011} C_VEL
LIN {X 0,Y 373.56,Z 551.76,A -85,B 0,C 180,E1 -12812.757,E2 -12812.757} C_VEL
LIN {X 0,Y 373.923,Z 538.366,A -85,B 0,C 180,E1 -12813.23,E2 -12813.23} C_VEL
LIN {X 0,Y 375.63,Z 456.614,A -85,B 0,C 180,E1 -12815.109,E2 -12815.109} C_VEL
LIN {X 0,Y 368.968,Z 437.524,A -85,B 0,C 180,E1 -12815.897,E2 -12815.897} C_VEL
LIN {X 0,Y 368.876,Z 437.534,A -85,B 0,C 180,E1 -12818.957,E2 -12818.957} C_VEL
LIN {X 0,Y 368.873,Z 437.535,A -85,B 0,C 180,E1 -12822.007,E2 -12822.007} C_VEL
LIN {X 0,Y 368.879,Z 437.532,A -85,B 0,C 180,E1 -12825.175,E2 -12825.175} C_VEL
LIN {X 0,Y 368.871,Z 437.537,A -85,B 0,C 180,E1 -12828.175,E2 -12828.175} C_VEL
LIN {X 0,Y 368.877,Z 437.532,A -85,B 0,C 180,E1 -12831.366,E2 -12831.366} C_VEL
LIN {X 0,Y 368.938,Z 437.525,A -85,B 0,C 180,E1 -12835.146,E2 -12835.146} C_VEL
LIN {X 0,Y 368.932,Z 437.526,A -85,B 0,C 180,E1 -12839.046,E2 -12839.046} C_VEL
LIN {X 0,Y 368.868,Z 437.536,A -85,B 0,C 180,E1 -12842.788,E2 -12842.788} C_VEL
LIN {X 0,Y 368.952,Z 437.53,A -85,B 0,C 180,E1 -12846.42,E2 -12846.42} C_VEL
LIN {X 0,Y 368.938,Z 437.526,A -85,B 0,C 180,E1 -12849.947,E2 -12849.947} C_VEL
LIN {X 0,Y 368.976,Z 437.52,A -85,B 0,C 180,E1 -12853.398,E2 -12853.398} C_VEL
LIN {X 0,Y 369.06,Z 437.513,A -85,B 0,C 180,E1 -12856.79,E2 -12856.79} C_VEL
LIN {X 0,Y 369.065,Z 437.512,A -85,B 0,C 180,E1 -12860.131,E2 -12860.131} C_VEL
LIN {X 0,Y 369.163,Z 437.497,A -85,B 0,C 180,E1 -12863.441,E2 -12863.441} C_VEL
LIN {X 0,Y 369.315,Z 437.478,A -85,B 0,C 180,E1 -12867.818,E2 -12867.818} C_VEL
LIN {X 0,Y 369.431,Z 437.465,A -85,B 0,C 180,E1 -12870,E2 -12870} C_VEL
